(* PLC project Error Translations, Hydac Systems GmbH PdtCodeBuilder.dll 1.2.7.80 *)
(* stored: companyURL http://www.hydac.com/, contentDescription This content was automatically generated. Please do not edit., creationDateTime 2025-04-18T16:40:50.760 *)

TYPE _eDm1ErrorText : (txt_Err_Spn1000_Fmi31_FmiExt255 := 0, txt_Err_Spn1001_Fmi31_FmiExt255 := 1, txt_Err_Spn1002_Fmi31_FmiExt255 := 2, txt_Err_Spn1003_Fmi31_FmiExt255 := 3, txt_Err_Spn1004_Fmi31_FmiExt255 := 4, txt_Err_Spn1005_Fmi31_FmiExt255 := 5, txt_Err_Spn1006_Fmi31_FmiExt255 := 6, txt_Err_Spn1007_Fmi31_FmiExt255 := 7, txt_Err_Spn1008_Fmi31_FmiExt255 := 8, txt_Err_Spn1009_Fmi31_FmiExt255 := 9, txt_Err_Spn1010_Fmi31_FmiExt255 := 10, txt_Err_Spn1011_Fmi31_FmiExt255 := 11, txt_Err_Spn1012_Fmi31_FmiExt255 := 12, txt_Err_Spn1013_Fmi31_FmiExt255 := 13, txt_Err_Spn1014_Fmi31_FmiExt255 := 14, txt_Err_Spn1015_Fmi31_FmiExt255 := 15, txt_Err_Spn1016_Fmi31_FmiExt255 := 16, txt_Err_Spn1017_Fmi31_FmiExt255 := 17, txt_Err_Spn1018_Fmi31_FmiExt255 := 18, txt_Err_Spn1019_Fmi31_FmiExt255 := 19, txt_Err_Spn1020_Fmi31_FmiExt255 := 20, txt_Err_Spn1021_Fmi31_FmiExt255 := 21, txt_Err_Spn1022_Fmi31_FmiExt255 := 22, txt_Err_Spn1023_Fmi31_FmiExt255 := 23, txt_Err_Spn1024_Fmi31_FmiExt255 := 24, txt_Err_Spn1031_Fmi31_FmiExt255 := 25, txt_Err_Spn1032_Fmi31_FmiExt255 := 26, txt_Err_Spn1033_Fmi31_FmiExt255 := 27, txt_Err_Spn1034_Fmi31_FmiExt255 := 28, txt_Err_Spn1035_Fmi31_FmiExt255 := 29, txt_Err_Spn1036_Fmi31_FmiExt255 := 30, txt_Err_Spn1037_Fmi31_FmiExt255 := 31, txt_Err_Spn1038_Fmi31_FmiExt255 := 32, txt_Err_Spn1039_Fmi31_FmiExt255 := 33, txt_Err_Spn1040_Fmi31_FmiExt255 := 34, txt_Err_Spn1041_Fmi31_FmiExt255 := 35, txt_Err_Spn1042_Fmi31_FmiExt255 := 36, txt_Err_Spn1043_Fmi31_FmiExt255 := 37, txt_Err_Spn1044_Fmi31_FmiExt255 := 38, txt_Err_Spn1045_Fmi31_FmiExt255 := 39, txt_Err_Spn1046_Fmi31_FmiExt255 := 40, txt_Err_Spn1047_Fmi31_FmiExt255 := 41, txt_Err_Spn1048_Fmi31_FmiExt255 := 42, txt_Err_Spn1049_Fmi31_FmiExt255 := 43, txt_Err_Spn1051_Fmi31_FmiExt255 := 44, txt_Err_Spn1052_Fmi31_FmiExt255 := 45, txt_Err_Spn1053_Fmi31_FmiExt255 := 46, txt_Err_Spn1054_Fmi31_FmiExt255 := 47, txt_Err_Spn1055_Fmi31_FmiExt255 := 48, txt_Err_Spn1056_Fmi31_FmiExt255 := 49, txt_Err_Spn1057_Fmi31_FmiExt255 := 50, txt_Err_Spn1058_Fmi31_FmiExt255 := 51, txt_Err_Spn1059_Fmi31_FmiExt255 := 52, txt_Err_Spn1060_Fmi31_FmiExt255 := 53, txt_Err_Spn1063_Fmi31_FmiExt255 := 54, txt_Err_Spn1064_Fmi31_FmiExt255 := 55, txt_Err_Spn1065_Fmi31_FmiExt255 := 56, txt_Err_Spn1066_Fmi31_FmiExt255 := 57, txt_Err_Spn1067_Fmi31_FmiExt255 := 58, txt_Err_Spn1068_Fmi31_FmiExt255 := 59, txt_Err_Spn1069_Fmi31_FmiExt255 := 60, txt_Err_Spn1070_Fmi31_FmiExt255 := 61, txt_Err_Spn1071_Fmi31_FmiExt255 := 62, txt_Err_Spn1072_Fmi31_FmiExt255 := 63, txt_Err_Spn1073_Fmi31_FmiExt255 := 64, txt_Err_Spn1074_Fmi31_FmiExt255 := 65, txt_Err_Spn1075_Fmi31_FmiExt255 := 66, txt_Err_Spn1082_Fmi31_FmiExt255 := 67, txt_Err_Spn1083_Fmi31_FmiExt255 := 68, txt_Err_Spn1084_Fmi31_FmiExt255 := 69, txt_Err_Spn1102_Fmi31_FmiExt255 := 70, txt_Err_Spn1103_Fmi31_FmiExt255 := 71, txt_Err_Spn1104_Fmi31_FmiExt255 := 72, txt_Err_Spn1105_Fmi31_FmiExt255 := 73, txt_Err_Spn1106_Fmi31_FmiExt255 := 74, txt_Err_Spn1107_Fmi31_FmiExt255 := 75, txt_Err_Spn1108_Fmi31_FmiExt255 := 76, txt_Err_Spn1109_Fmi31_FmiExt255 := 77, txt_Err_Spn1110_Fmi31_FmiExt255 := 78, txt_Err_Spn1111_Fmi31_FmiExt255 := 79, txt_Err_Spn1112_Fmi31_FmiExt255 := 80, txt_Err_Spn1113_Fmi31_FmiExt255 := 81, txt_Err_Spn1114_Fmi31_FmiExt255 := 82, txt_Err_Spn1115_Fmi31_FmiExt255 := 83, txt_Err_Spn1116_Fmi31_FmiExt255 := 84, txt_Err_Spn1117_Fmi31_FmiExt255 := 85, txt_Err_Spn1118_Fmi31_FmiExt255 := 86, txt_Err_Spn1119_Fmi31_FmiExt255 := 87, txt_Err_Spn1153_Fmi31_FmiExt255 := 88, txt_Err_Spn1154_Fmi31_FmiExt255 := 89, txt_Err_Spn1155_Fmi31_FmiExt255 := 90, txt_Err_Spn1156_Fmi31_FmiExt255 := 91, txt_Err_Spn1157_Fmi31_FmiExt255 := 92, txt_Err_Spn1158_Fmi31_FmiExt255 := 93, txt_Err_Spn1159_Fmi31_FmiExt255 := 94, txt_Err_Spn1160_Fmi31_FmiExt255 := 95, txt_Err_Spn1161_Fmi31_FmiExt255 := 96, txt_Err_Spn1162_Fmi31_FmiExt255 := 97, txt_Err_Spn1163_Fmi31_FmiExt255 := 98, txt_Err_Spn1164_Fmi31_FmiExt255 := 99, txt_Err_Spn1165_Fmi31_FmiExt255 := 100, txt_Err_Spn1166_Fmi31_FmiExt255 := 101, txt_Err_Spn1167_Fmi31_FmiExt255 := 102, txt_Err_Spn1168_Fmi31_FmiExt255 := 103, txt_Err_Spn1173_Fmi31_FmiExt255 := 104, txt_Err_Spn1174_Fmi31_FmiExt255 := 105, txt_Err_Spn1175_Fmi31_FmiExt255 := 106, txt_Err_Spn1176_Fmi31_FmiExt255 := 107, txt_Err_Spn1177_Fmi31_FmiExt255 := 108, txt_Err_Spn1178_Fmi31_FmiExt255 := 109, txt_Err_Spn1179_Fmi31_FmiExt255 := 110, txt_Err_Spn1180_Fmi31_FmiExt255 := 111, txt_Err_Spn1181_Fmi31_FmiExt255 := 112, txt_Err_Spn1182_Fmi31_FmiExt255 := 113, txt_Err_Spn1183_Fmi31_FmiExt255 := 114, txt_Err_Spn1184_Fmi31_FmiExt255 := 115, txt_Err_Spn1185_Fmi31_FmiExt255 := 116, txt_Err_Spn1186_Fmi31_FmiExt255 := 117, txt_Err_Spn1187_Fmi31_FmiExt255 := 118, txt_Err_Spn1188_Fmi31_FmiExt255 := 119, txt_Err_Spn1189_Fmi31_FmiExt255 := 120, txt_Err_Spn1190_Fmi31_FmiExt255 := 121, txt_Err_Spn1203_Fmi31_FmiExt255 := 122, txt_Err_Spn1205_Fmi31_FmiExt255 := 123, txt_Err_Spn1209_Fmi31_FmiExt255 := 124, txt_Err_Spn1210_Fmi31_FmiExt255 := 125, txt_Err_Spn1211_Fmi31_FmiExt255 := 126, txt_Err_Spn1212_Fmi31_FmiExt255 := 127, txt_Err_Spn1213_Fmi31_FmiExt255 := 128, txt_Err_Spn1214_Fmi31_FmiExt255 := 129, txt_Err_Spn1215_Fmi31_FmiExt255 := 130, txt_Err_Spn1216_Fmi31_FmiExt255 := 131, txt_Err_Spn1217_Fmi31_FmiExt255 := 132, txt_Err_Spn1218_Fmi31_FmiExt255 := 133, txt_Err_Spn1219_Fmi31_FmiExt255 := 134, txt_Err_Spn1220_Fmi31_FmiExt255 := 135, txt_Err_Spn1221_Fmi31_FmiExt255 := 136, txt_Err_Spn1222_Fmi31_FmiExt255 := 137, txt_Err_Spn1223_Fmi31_FmiExt255 := 138, txt_Err_Spn1224_Fmi31_FmiExt255 := 139, txt_Err_Spn1225_Fmi31_FmiExt255 := 140, txt_Err_Spn1226_Fmi31_FmiExt255 := 141, txt_Err_Spn1229_Fmi31_FmiExt255 := 142, txt_Err_Spn1230_Fmi31_FmiExt255 := 143, txt_Err_Spn1231_Fmi31_FmiExt255 := 144, txt_Err_Spn1232_Fmi31_FmiExt255 := 145, txt_Err_Spn1233_Fmi31_FmiExt255 := 146, txt_Err_Spn1234_Fmi31_FmiExt255 := 147, txt_Err_Spn1235_Fmi31_FmiExt255 := 148, txt_Err_Spn1236_Fmi31_FmiExt255 := 149, txt_Err_Spn1237_Fmi31_FmiExt255 := 150, txt_Err_Spn1238_Fmi31_FmiExt255 := 151, txt_Err_Spn1239_Fmi31_FmiExt255 := 152, txt_Err_Spn1240_Fmi31_FmiExt255 := 153, txt_Err_Spn1241_Fmi31_FmiExt255 := 154, txt_Err_Spn1242_Fmi31_FmiExt255 := 155, txt_Err_Spn1243_Fmi31_FmiExt255 := 156, txt_Err_Spn1244_Fmi31_FmiExt255 := 157, txt_Err_Spn1245_Fmi31_FmiExt255 := 158, txt_Err_Spn1246_Fmi31_FmiExt255 := 159, txt_Err_Spn1247_Fmi31_FmiExt255 := 160, txt_Err_Spn1253_Fmi31_FmiExt255 := 161, txt_Err_Spn1254_Fmi31_FmiExt255 := 162, txt_Err_Spn1255_Fmi31_FmiExt255 := 163, txt_Err_Spn1256_Fmi31_FmiExt255 := 164, txt_Err_Spn1257_Fmi31_FmiExt255 := 165, txt_Err_Spn1265_Fmi31_FmiExt255 := 166, txt_Err_Spn1266_Fmi31_FmiExt255 := 167, txt_Err_Spn1267_Fmi31_FmiExt255 := 168, txt_Err_Spn1268_Fmi31_FmiExt255 := 169, txt_Err_Spn1269_Fmi31_FmiExt255 := 170, txt_Err_Spn1277_Fmi31_FmiExt255 := 171, txt_Err_Spn1278_Fmi31_FmiExt255 := 172, txt_Err_Spn1279_Fmi31_FmiExt255 := 173, txt_Err_Spn1280_Fmi31_FmiExt255 := 174, txt_Err_Spn1281_Fmi31_FmiExt255 := 175, txt_Err_Spn1287_Fmi31_FmiExt255 := 176, txt_Err_Spn1288_Fmi31_FmiExt255 := 177, txt_Err_Spn1289_Fmi31_FmiExt255 := 178, txt_Err_Spn1290_Fmi31_FmiExt255 := 179, txt_Err_Spn1291_Fmi31_FmiExt255 := 180, txt_Err_Spn1292_Fmi31_FmiExt255 := 181, txt_Err_Spn1293_Fmi31_FmiExt255 := 182, txt_Err_Spn1294_Fmi31_FmiExt255 := 183, txt_Err_Spn1295_Fmi31_FmiExt255 := 184, txt_Err_Spn1296_Fmi31_FmiExt255 := 185, txt_Err_Spn1297_Fmi31_FmiExt255 := 186, txt_Err_Spn1298_Fmi31_FmiExt255 := 187, txt_Err_Spn1299_Fmi31_FmiExt255 := 188, txt_Err_Spn1300_Fmi31_FmiExt255 := 189, txt_Err_Spn1301_Fmi31_FmiExt255 := 190, txt_Err_Spn1302_Fmi31_FmiExt255 := 191, txt_Err_Spn1303_Fmi31_FmiExt255 := 192, txt_Err_Spn1304_Fmi31_FmiExt255 := 193, txt_Err_Spn1305_Fmi31_FmiExt255 := 194, txt_Err_Spn1306_Fmi31_FmiExt255 := 195, txt_Err_Spn1307_Fmi31_FmiExt255 := 196, txt_Err_Spn1308_Fmi31_FmiExt255 := 197, txt_Err_Spn1309_Fmi31_FmiExt255 := 198, txt_Err_Spn1310_Fmi31_FmiExt255 := 199, txt_Err_Spn1311_Fmi31_FmiExt255 := 200, txt_Err_Spn1312_Fmi31_FmiExt255 := 201, txt_Err_Spn1313_Fmi31_FmiExt255 := 202, txt_Err_Spn1314_Fmi31_FmiExt255 := 203, txt_Err_Spn1315_Fmi31_FmiExt255 := 204, txt_Err_Spn1316_Fmi31_FmiExt255 := 205, txt_Err_Spn1317_Fmi31_FmiExt255 := 206, txt_Err_Spn1318_Fmi31_FmiExt255 := 207, txt_Err_Spn1319_Fmi31_FmiExt255 := 208, txt_Err_Spn1320_Fmi31_FmiExt255 := 209, txt_Err_Spn1321_Fmi31_FmiExt255 := 210, txt_Err_Spn1322_Fmi31_FmiExt255 := 211, txt_Err_Spn1339_Fmi31_FmiExt255 := 212, txt_Err_Spn1345_Fmi31_FmiExt255 := 213, txt_Err_Spn1346_Fmi31_FmiExt255 := 214, txt_Err_Spn1347_Fmi31_FmiExt255 := 215, txt_Err_Spn1348_Fmi31_FmiExt255 := 216, txt_Err_Spn1349_Fmi31_FmiExt255 := 217, txt_Err_Spn1350_Fmi31_FmiExt255 := 218, txt_Err_Spn1351_Fmi31_FmiExt255 := 219, txt_Err_Spn1352_Fmi31_FmiExt255 := 220, txt_Err_Spn1353_Fmi31_FmiExt255 := 221, txt_Err_Spn1356_Fmi31_FmiExt255 := 222, txt_Err_Spn1357_Fmi31_FmiExt255 := 223, txt_Err_Spn1358_Fmi31_FmiExt255 := 224, txt_Err_Spn1359_Fmi31_FmiExt255 := 225, txt_Err_Spn1360_Fmi31_FmiExt255 := 226, txt_Err_Spn1361_Fmi31_FmiExt255 := 227, txt_Err_Spn1362_Fmi31_FmiExt255 := 228, txt_Err_Spn1363_Fmi31_FmiExt255 := 229, txt_Err_Spn1364_Fmi31_FmiExt255 := 230, txt_Err_Spn1365_Fmi31_FmiExt255 := 231, txt_Err_Spn1366_Fmi31_FmiExt255 := 232, txt_Err_Spn1367_Fmi31_FmiExt255 := 233, txt_Err_Spn1368_Fmi31_FmiExt255 := 234, txt_Err_Spn1369_Fmi31_FmiExt255 := 235, txt_Err_Spn1370_Fmi31_FmiExt255 := 236, txt_Err_Spn1371_Fmi31_FmiExt255 := 237, txt_Err_Spn1372_Fmi31_FmiExt255 := 238, txt_Err_Spn1373_Fmi31_FmiExt255 := 239, txt_Err_Spn1439_Fmi31_FmiExt255 := 240, txt_Err_Spn1440_Fmi31_FmiExt255 := 241, txt_Err_Spn1441_Fmi31_FmiExt255 := 242, txt_Err_Spn1442_Fmi31_FmiExt255 := 243, txt_Err_Spn1443_Fmi31_FmiExt255 := 244, txt_Err_Spn1449_Fmi31_FmiExt255 := 245, txt_Err_Spn1450_Fmi31_FmiExt255 := 246, txt_Err_Spn1451_Fmi31_FmiExt255 := 247, txt_Err_Spn1452_Fmi31_FmiExt255 := 248, txt_Err_Spn1453_Fmi31_FmiExt255 := 249, txt_Err_Spn1459_Fmi31_FmiExt255 := 250, txt_Err_Spn1460_Fmi31_FmiExt255 := 251, txt_Err_Spn1461_Fmi31_FmiExt255 := 252, txt_Err_Spn1462_Fmi31_FmiExt255 := 253, txt_Err_Spn1463_Fmi31_FmiExt255 := 254, txt_Err_Spn1469_Fmi31_FmiExt255 := 255, txt_Err_Spn1470_Fmi31_FmiExt255 := 256, txt_Err_Spn1471_Fmi31_FmiExt255 := 257, txt_Err_Spn1472_Fmi31_FmiExt255 := 258, txt_Err_Spn1473_Fmi31_FmiExt255 := 259, txt_Err_Spn1479_Fmi31_FmiExt255 := 260, txt_Err_Spn1480_Fmi31_FmiExt255 := 261, txt_Err_Spn1481_Fmi31_FmiExt255 := 262, txt_Err_Spn1482_Fmi31_FmiExt255 := 263, txt_Err_Spn1483_Fmi31_FmiExt255 := 264, txt_Err_Spn1536_Fmi31_FmiExt255 := 265, txt_Err_Spn1542_Fmi31_FmiExt255 := 266, txt_Err_Spn1543_Fmi31_FmiExt255 := 267, txt_Err_Spn1554_Fmi31_FmiExt255 := 268, txt_Err_Spn1566_Fmi31_FmiExt255 := 269, txt_Err_Spn1567_Fmi31_FmiExt255 := 270, txt_Err_Spn1568_Fmi31_FmiExt255 := 271, txt_Err_Spn1569_Fmi31_FmiExt255 := 272, txt_Err_Spn1570_Fmi31_FmiExt255 := 273, txt_Err_Spn1571_Fmi31_FmiExt255 := 274, txt_Err_Spn1572_Fmi31_FmiExt255 := 275, txt_Err_Spn1573_Fmi31_FmiExt255 := 276, txt_Err_Spn1574_Fmi31_FmiExt255 := 277, txt_Err_Spn1575_Fmi31_FmiExt255 := 278, txt_Err_Spn1576_Fmi31_FmiExt255 := 279, txt_Err_Spn1577_Fmi31_FmiExt255 := 280, txt_Err_Spn1578_Fmi31_FmiExt255 := 281, txt_Err_Spn1579_Fmi31_FmiExt255 := 282, txt_Err_Spn1580_Fmi31_FmiExt255 := 283, txt_Err_Spn1581_Fmi31_FmiExt255 := 284, txt_Err_Spn1582_Fmi31_FmiExt255 := 285, txt_Err_Spn1583_Fmi31_FmiExt255 := 286, txt_Err_Spn1584_Fmi31_FmiExt255 := 287, txt_Err_Spn1585_Fmi31_FmiExt255 := 288, txt_Err_Spn1586_Fmi31_FmiExt255 := 289, txt_Err_Spn1587_Fmi31_FmiExt255 := 290, txt_Err_Spn1588_Fmi31_FmiExt255 := 291, txt_Err_Spn1589_Fmi31_FmiExt255 := 292, txt_Err_Spn1590_Fmi31_FmiExt255 := 293, txt_Err_Spn1591_Fmi31_FmiExt255 := 294, txt_Err_Spn1592_Fmi31_FmiExt255 := 295, txt_Err_Spn1593_Fmi31_FmiExt255 := 296, txt_Err_Spn1594_Fmi31_FmiExt255 := 297, txt_Err_Spn1595_Fmi31_FmiExt255 := 298, txt_Err_Spn1596_Fmi31_FmiExt255 := 299, txt_Err_Spn1597_Fmi31_FmiExt255 := 300, txt_Err_Spn1598_Fmi31_FmiExt255 := 301, txt_Err_Spn9000_Fmi3_FmiExt255 := 302, txt_Err_Spn9001_Fmi4_FmiExt255 := 303, txt_Err_Spn9002_Fmi24_FmiExt255 := 304, txt_Err_Spn9003_Fmi12_FmiExt255 := 305, txt_Err_Spn9004_Fmi3_FmiExt255 := 306, txt_Err_Spn9005_Fmi4_FmiExt255 := 307, txt_Err_Spn9006_Fmi24_FmiExt255 := 308, txt_Err_Spn9007_Fmi12_FmiExt255 := 309, txt_Err_Spn9008_Fmi3_FmiExt255 := 310, txt_Err_Spn9009_Fmi4_FmiExt255 := 311, txt_Err_Spn9010_Fmi24_FmiExt255 := 312, txt_Err_Spn9011_Fmi12_FmiExt255 := 313, txt_Err_Spn9012_Fmi31_FmiExt255 := 314, txt_Err_Spn9013_Fmi31_FmiExt255 := 315, txt_Err_Spn9014_Fmi31_FmiExt255 := 316, txt_Err_Spn9015_Fmi31_FmiExt255 := 317, txt_Err_Spn9016_Fmi31_FmiExt255 := 318, txt_Err_Spn9017_Fmi31_FmiExt255 := 319, txt_Err_Spn9018_Fmi31_FmiExt255 := 320, txt_Err_Spn9019_Fmi31_FmiExt255 := 321, txt_Err_Spn9020_Fmi31_FmiExt255 := 322, txt_Err_Spn9021_Fmi31_FmiExt255 := 323, txt_Err_Spn9022_Fmi31_FmiExt255 := 324, txt_Err_Spn9023_Fmi31_FmiExt255 := 325, txt_Err_Spn9024_Fmi31_FmiExt255 := 326, txt_Err_Spn9025_Fmi31_FmiExt255 := 327, txt_Err_Spn9026_Fmi31_FmiExt255 := 328, txt_Err_Spn9027_Fmi31_FmiExt255 := 329, txt_Err_Spn9028_Fmi31_FmiExt255 := 330, txt_Err_Spn9029_Fmi31_FmiExt255 := 331, txt_Err_Spn9030_Fmi31_FmiExt255 := 332, txt_Err_Spn9031_Fmi31_FmiExt255 := 333, txt_Err_Spn9032_Fmi31_FmiExt255 := 334, txt_Err_Spn9033_Fmi31_FmiExt255 := 335, txt_Err_Spn9034_Fmi31_FmiExt255 := 336, txt_Err_Spn9035_Fmi31_FmiExt255 := 337, txt_Err_Spn9036_Fmi31_FmiExt255 := 338, txt_Err_Spn9037_Fmi31_FmiExt255 := 339, txt_Err_Spn9038_Fmi31_FmiExt255 := 340, txt_Err_Spn9039_Fmi31_FmiExt255 := 341, txt_Err_Spn9040_Fmi31_FmiExt255 := 342, txt_Err_Spn9041_Fmi31_FmiExt255 := 343, txt_Err_Spn9042_Fmi31_FmiExt255 := 344, txt_Err_Spn9043_Fmi31_FmiExt255 := 345, txt_Err_Spn9044_Fmi31_FmiExt255 := 346, txt_Err_Spn9045_Fmi31_FmiExt255 := 347, txt_Err_Spn9046_Fmi31_FmiExt255 := 348, txt_Err_Spn9047_Fmi31_FmiExt255 := 349, txt_Err_Spn9048_Fmi3_FmiExt255 := 350, txt_Err_Spn9049_Fmi4_FmiExt255 := 351, txt_Err_Spn9050_Fmi24_FmiExt255 := 352, txt_Err_Spn9051_Fmi12_FmiExt255 := 353, txt_Err_Spn9052_Fmi31_FmiExt255 := 354, txt_Err_Spn9053_Fmi31_FmiExt255 := 355, txt_Err_Spn9054_Fmi31_FmiExt255 := 356, txt_Err_Spn9055_Fmi31_FmiExt255 := 357, txt_Err_Spn9056_Fmi31_FmiExt255 := 358, txt_Err_Spn9057_Fmi31_FmiExt255 := 359, txt_Err_Spn9058_Fmi31_FmiExt255 := 360, txt_Err_Spn9059_Fmi31_FmiExt255 := 361, txt_Err_Spn9060_Fmi31_FmiExt255 := 362, txt_Err_Spn9061_Fmi31_FmiExt255 := 363, txt_Err_Spn9062_Fmi31_FmiExt255 := 364, txt_Err_Spn9063_Fmi31_FmiExt255 := 365, txt_Err_Spn9064_Fmi3_FmiExt255 := 366, txt_Err_Spn9065_Fmi4_FmiExt255 := 367, txt_Err_Spn9066_Fmi24_FmiExt255 := 368, txt_Err_Spn9067_Fmi12_FmiExt255 := 369, txt_Err_Spn9068_Fmi31_FmiExt255 := 370, txt_Err_Spn9069_Fmi31_FmiExt255 := 371, txt_Err_Spn9070_Fmi31_FmiExt255 := 372, txt_Err_Spn9071_Fmi31_FmiExt255 := 373, txt_Err_Spn9072_Fmi31_FmiExt255 := 374, txt_Err_Spn9073_Fmi31_FmiExt255 := 375, txt_Err_Spn9074_Fmi31_FmiExt255 := 376, txt_Err_Spn9075_Fmi31_FmiExt255 := 377, txt_Err_Spn9076_Fmi31_FmiExt255 := 378, txt_Err_Spn9077_Fmi31_FmiExt255 := 379, txt_Err_Spn9078_Fmi31_FmiExt255 := 380, txt_Err_Spn9079_Fmi31_FmiExt255 := 381, txt_Err_Spn9080_Fmi31_FmiExt255 := 382, txt_Err_Spn9081_Fmi31_FmiExt255 := 383, txt_Err_Spn9082_Fmi31_FmiExt255 := 384, txt_Err_Spn9083_Fmi31_FmiExt255 := 385, txt_Err_Spn9084_Fmi31_FmiExt255 := 386, txt_Err_Spn9085_Fmi31_FmiExt255 := 387, txt_Err_Spn9086_Fmi31_FmiExt255 := 388, txt_Err_Spn9087_Fmi31_FmiExt255 := 389, txt_Err_Spn9088_Fmi31_FmiExt255 := 390, txt_Err_Spn9089_Fmi31_FmiExt255 := 391, txt_Err_Spn9090_Fmi31_FmiExt255 := 392, txt_Err_Spn9091_Fmi31_FmiExt255 := 393, txt_Err_Spn9092_Fmi31_FmiExt255 := 394, txt_Err_Spn9093_Fmi31_FmiExt255 := 395, txt_Err_Spn9094_Fmi31_FmiExt255 := 396, txt_Err_Spn9095_Fmi31_FmiExt255 := 397, txt_Err_Spn9096_Fmi31_FmiExt255 := 398, txt_Err_Spn9097_Fmi31_FmiExt255 := 399, txt_Err_Spn9098_Fmi31_FmiExt255 := 400, txt_Err_Spn9099_Fmi31_FmiExt255 := 401, txt_Err_Spn9100_Fmi31_FmiExt255 := 402, txt_Err_Spn9101_Fmi31_FmiExt255 := 403, txt_Err_Spn9102_Fmi31_FmiExt255 := 404, txt_Err_Spn9103_Fmi31_FmiExt255 := 405, txt_Err_Spn9104_Fmi31_FmiExt255 := 406, txt_Err_Spn9105_Fmi31_FmiExt255 := 407, txt_Err_Spn9106_Fmi31_FmiExt255 := 408, txt_Err_Spn9107_Fmi31_FmiExt255 := 409, txt_Err_Spn9108_Fmi31_FmiExt255 := 410, txt_Err_Spn9109_Fmi31_FmiExt255 := 411, txt_Err_Spn9110_Fmi31_FmiExt255 := 412, txt_Err_Spn9111_Fmi31_FmiExt255 := 413, txt_Err_Spn9112_Fmi31_FmiExt255 := 414, txt_Err_Spn9113_Fmi31_FmiExt255 := 415, txt_Err_Spn9114_Fmi31_FmiExt255 := 416, txt_Err_Spn9115_Fmi31_FmiExt255 := 417, txt_Err_Spn9116_Fmi31_FmiExt255 := 418, txt_Err_Spn9117_Fmi31_FmiExt255 := 419, txt_Err_Spn9118_Fmi31_FmiExt255 := 420, txt_Err_Spn9119_Fmi31_FmiExt255 := 421, txt_Err_Spn9120_Fmi31_FmiExt255 := 422, txt_Err_Spn9121_Fmi31_FmiExt255 := 423, txt_Err_Spn9122_Fmi31_FmiExt255 := 424, txt_Err_Spn9123_Fmi31_FmiExt255 := 425, txt_Err_Spn9124_Fmi31_FmiExt255 := 426, txt_Err_Spn9125_Fmi31_FmiExt255 := 427, txt_Err_Spn9126_Fmi31_FmiExt255 := 428, txt_Err_Spn9127_Fmi31_FmiExt255 := 429, txt_Err_Spn9128_Fmi31_FmiExt255 := 430, txt_Err_Spn9129_Fmi31_FmiExt255 := 431, txt_Err_Spn9130_Fmi31_FmiExt255 := 432, txt_Err_Spn9131_Fmi31_FmiExt255 := 433, txt_Err_Spn9132_Fmi31_FmiExt255 := 434, txt_Err_Spn9133_Fmi31_FmiExt255 := 435, txt_Err_Spn9134_Fmi31_FmiExt255 := 436, txt_Err_Spn9135_Fmi31_FmiExt255 := 437, txt_Err_Spn9136_Fmi31_FmiExt255 := 438, txt_Err_Spn9137_Fmi31_FmiExt255 := 439, txt_Err_Spn9138_Fmi31_FmiExt255 := 440, txt_Err_Spn9139_Fmi31_FmiExt255 := 441, txt_Err_Spn9140_Fmi31_FmiExt255 := 442, txt_Err_Spn9141_Fmi31_FmiExt255 := 443, txt_Err_Spn9142_Fmi31_FmiExt255 := 444, txt_Err_Spn9143_Fmi31_FmiExt255 := 445, txt_Err_Spn9144_Fmi31_FmiExt255 := 446, txt_Err_Spn9145_Fmi31_FmiExt255 := 447, txt_Err_Spn9146_Fmi31_FmiExt255 := 448, txt_Err_Spn9147_Fmi31_FmiExt255 := 449, txt_Err_Spn9148_Fmi31_FmiExt255 := 450, txt_Err_Spn9149_Fmi31_FmiExt255 := 451, txt_Err_Spn9150_Fmi31_FmiExt255 := 452, txt_Err_Spn9151_Fmi31_FmiExt255 := 453, txt_Err_Spn9152_Fmi31_FmiExt255 := 454, txt_Err_Spn9153_Fmi31_FmiExt255 := 455, txt_Err_Spn9154_Fmi31_FmiExt255 := 456, txt_Err_Spn9155_Fmi31_FmiExt255 := 457, txt_Err_Spn9156_Fmi31_FmiExt255 := 458, txt_Err_Spn9157_Fmi31_FmiExt255 := 459, txt_Err_Spn9158_Fmi31_FmiExt255 := 460, txt_Err_Spn9159_Fmi31_FmiExt255 := 461, txt_Err_Spn9160_Fmi31_FmiExt255 := 462, txt_Err_Spn9161_Fmi31_FmiExt255 := 463, txt_Err_Spn9162_Fmi31_FmiExt255 := 464, txt_Err_Spn9163_Fmi31_FmiExt255 := 465, txt_Err_Spn9164_Fmi31_FmiExt255 := 466, txt_Err_Spn9165_Fmi31_FmiExt255 := 467, txt_Err_Spn9166_Fmi31_FmiExt255 := 468, txt_Err_Spn9167_Fmi31_FmiExt255 := 469, txt_Err_Spn9168_Fmi31_FmiExt255 := 470, txt_Err_Spn9169_Fmi31_FmiExt255 := 471, txt_Err_Spn9170_Fmi31_FmiExt255 := 472, txt_Err_Spn9171_Fmi31_FmiExt255 := 473, txt_Err_Spn9172_Fmi31_FmiExt255 := 474, txt_Err_Spn9173_Fmi3_FmiExt255 := 475, txt_Err_Spn9174_Fmi4_FmiExt255 := 476, txt_Err_Spn9175_Fmi24_FmiExt255 := 477, txt_Err_Spn9176_Fmi12_FmiExt255 := 478, txt_Err_Spn9177_Fmi31_FmiExt255 := 479, txt_Err_Spn9178_Fmi31_FmiExt255 := 480, txt_Err_Spn9179_Fmi31_FmiExt255 := 481, txt_Err_Spn9180_Fmi31_FmiExt255 := 482, txt_Err_Spn9181_Fmi31_FmiExt255 := 483, txt_Err_Spn9182_Fmi31_FmiExt255 := 484, txt_Err_Spn9183_Fmi31_FmiExt255 := 485, txt_Err_Spn9184_Fmi31_FmiExt255 := 486, txt_Err_Spn9185_Fmi31_FmiExt255 := 487, txt_Err_Spn9186_Fmi31_FmiExt255 := 488, txt_Err_Spn9187_Fmi31_FmiExt255 := 489, txt_Err_Spn9188_Fmi31_FmiExt255 := 490, txt_Err_Spn9189_Fmi31_FmiExt255 := 491, txt_Err_Spn9190_Fmi31_FmiExt255 := 492, txt_Err_Spn9191_Fmi31_FmiExt255 := 493, txt_Err_Spn9192_Fmi31_FmiExt255 := 494, txt_Err_Spn9193_Fmi31_FmiExt255 := 495, txt_Err_Spn9194_Fmi31_FmiExt255 := 496, txt_Err_Spn9195_Fmi31_FmiExt255 := 497, txt_Err_Spn9196_Fmi31_FmiExt255 := 498, txt_Err_Spn9197_Fmi31_FmiExt255 := 499, txt_Err_Spn9198_Fmi31_FmiExt255 := 500, txt_Err_Spn9199_Fmi31_FmiExt255 := 501, txt_Err_Spn9200_Fmi31_FmiExt255 := 502, txt_Err_Spn9201_Fmi31_FmiExt255 := 503, txt_Err_Spn9202_Fmi31_FmiExt255 := 504, txt_Err_Spn9203_Fmi31_FmiExt255 := 505, txt_Err_Spn9204_Fmi31_FmiExt255 := 506, txt_Err_Spn9205_Fmi31_FmiExt255 := 507, txt_Err_Spn9206_Fmi31_FmiExt255 := 508, txt_Err_Spn9207_Fmi31_FmiExt255 := 509, txt_Err_Spn9208_Fmi31_FmiExt255 := 510, txt_Err_Spn9209_Fmi31_FmiExt255 := 511, txt_Err_Spn9210_Fmi31_FmiExt255 := 512, txt_Err_Spn9211_Fmi31_FmiExt255 := 513, txt_Err_Spn9212_Fmi31_FmiExt255 := 514, txt_Err_Spn9213_Fmi31_FmiExt255 := 515, txt_Err_Spn9214_Fmi31_FmiExt255 := 516, txt_Err_Spn9215_Fmi31_FmiExt255 := 517, txt_Err_Spn9216_Fmi31_FmiExt255 := 518, txt_Err_Spn9217_Fmi31_FmiExt255 := 519, txt_Err_Spn9218_Fmi31_FmiExt255 := 520, txt_Err_Spn9219_Fmi31_FmiExt255 := 521, txt_Err_Spn9220_Fmi31_FmiExt255 := 522, txt_Err_Spn9221_Fmi31_FmiExt255 := 523, txt_Err_Spn9222_Fmi31_FmiExt255 := 524, txt_Err_Spn9223_Fmi31_FmiExt255 := 525, txt_Err_Spn9224_Fmi31_FmiExt255 := 526, txt_Err_Spn9225_Fmi31_FmiExt255 := 527, txt_Err_Spn9226_Fmi31_FmiExt255 := 528, txt_Err_Spn9227_Fmi31_FmiExt255 := 529, txt_Err_Spn9228_Fmi31_FmiExt255 := 530, txt_Err_Spn9237_Fmi31_FmiExt255 := 531, txt_Err_Spn9238_Fmi31_FmiExt255 := 532, txt_Err_Spn9239_Fmi31_FmiExt255 := 533, txt_Err_Spn9240_Fmi31_FmiExt255 := 534, txt_Err_Spn9241_Fmi31_FmiExt255 := 535, txt_Err_Spn9242_Fmi31_FmiExt255 := 536, txt_Err_Spn9243_Fmi31_FmiExt255 := 537, txt_Err_Spn9244_Fmi31_FmiExt255 := 538, txt_Err_Spn9245_Fmi31_FmiExt255 := 539, txt_Err_Spn9246_Fmi3_FmiExt255 := 540, txt_Err_Spn9247_Fmi4_FmiExt255 := 541, txt_Err_Spn9248_Fmi24_FmiExt255 := 542, txt_Err_Spn9249_Fmi12_FmiExt255 := 543, txt_Err_Spn9250_Fmi3_FmiExt255 := 544, txt_Err_Spn9251_Fmi4_FmiExt255 := 545, txt_Err_Spn9252_Fmi24_FmiExt255 := 546, txt_Err_Spn9253_Fmi12_FmiExt255 := 547, txt_Err_Spn9254_Fmi31_FmiExt255 := 548, txt_Err_Spn9255_Fmi31_FmiExt255 := 549, txt_Err_Spn9256_Fmi31_FmiExt255 := 550, txt_Err_Spn9257_Fmi31_FmiExt255 := 551, txt_Err_Spn9258_Fmi31_FmiExt255 := 552, txt_Err_Spn9259_Fmi31_FmiExt255 := 553, txt_Err_Spn9260_Fmi31_FmiExt255 := 554, txt_Err_Spn9261_Fmi31_FmiExt255 := 555, txt_Err_Spn9262_Fmi31_FmiExt255 := 556, txt_Err_Spn9263_Fmi31_FmiExt255 := 557, txt_Err_Spn9264_Fmi31_FmiExt255 := 558, txt_Err_Spn9265_Fmi31_FmiExt255 := 559, txt_Err_Spn9266_Fmi31_FmiExt255 := 560, txt_Err_Spn9267_Fmi31_FmiExt255 := 561, txt_Err_Spn9268_Fmi31_FmiExt255 := 562, txt_Err_Spn9269_Fmi31_FmiExt255 := 563, txt_Err_Spn9270_Fmi31_FmiExt255 := 564, txt_Err_Spn9271_Fmi31_FmiExt255 := 565, txt_Err_Spn9272_Fmi31_FmiExt255 := 566, txt_Err_Spn9273_Fmi31_FmiExt255 := 567, txt_Err_Spn9274_Fmi31_FmiExt255 := 568, txt_Err_Spn9275_Fmi31_FmiExt255 := 569, txt_Err_Spn9276_Fmi31_FmiExt255 := 570, txt_Err_Spn9277_Fmi31_FmiExt255 := 571, txt_Err_Spn9278_Fmi31_FmiExt255 := 572, txt_Err_Spn9279_Fmi31_FmiExt255 := 573, txt_Err_Spn9280_Fmi31_FmiExt255 := 574, txt_Err_Spn9281_Fmi31_FmiExt255 := 575, txt_Err_Spn9282_Fmi31_FmiExt255 := 576, txt_Err_Spn9283_Fmi31_FmiExt255 := 577, txt_Err_Spn9284_Fmi31_FmiExt255 := 578, txt_Err_Spn9285_Fmi31_FmiExt255 := 579, txt_Err_Spn9286_Fmi31_FmiExt255 := 580, txt_Err_Spn9287_Fmi31_FmiExt255 := 581, txt_Err_Spn9288_Fmi31_FmiExt255 := 582, txt_Err_Spn9289_Fmi31_FmiExt255 := 583, txt_Err_Spn9290_Fmi31_FmiExt255 := 584, txt_Err_Spn9291_Fmi31_FmiExt255 := 585, txt_Err_Spn9292_Fmi31_FmiExt255 := 586, txt_Err_Spn9293_Fmi31_FmiExt255 := 587, txt_Err_Spn9294_Fmi31_FmiExt255 := 588, txt_Err_Spn9295_Fmi31_FmiExt255 := 589, txt_Err_Spn9296_Fmi31_FmiExt255 := 590, txt_Err_Spn9297_Fmi31_FmiExt255 := 591, txt_Err_Spn9298_Fmi31_FmiExt255 := 592, txt_Err_Spn9299_Fmi31_FmiExt255 := 593, txt_Err_Spn9300_Fmi31_FmiExt255 := 594, txt_Err_Spn9301_Fmi31_FmiExt255 := 595, txt_Err_Spn9302_Fmi31_FmiExt255 := 596, txt_Err_Spn9303_Fmi31_FmiExt255 := 597, txt_Err_Spn9304_Fmi31_FmiExt255 := 598, txt_Err_Spn9305_Fmi31_FmiExt255 := 599, txt_Err_Spn9306_Fmi31_FmiExt255 := 600, txt_Err_Spn9307_Fmi31_FmiExt255 := 601, txt_Err_Spn9308_Fmi31_FmiExt255 := 602, txt_Err_Spn9309_Fmi31_FmiExt255 := 603, txt_Err_Spn9310_Fmi31_FmiExt255 := 604, txt_Err_Spn9311_Fmi31_FmiExt255 := 605, txt_Err_Spn9312_Fmi31_FmiExt255 := 606, txt_Err_Spn9313_Fmi31_FmiExt255 := 607, txt_Err_Spn9314_Fmi31_FmiExt255 := 608, txt_Err_Spn9315_Fmi31_FmiExt255 := 609, txt_Err_Spn9316_Fmi31_FmiExt255 := 610, txt_Err_Spn9317_Fmi31_FmiExt255 := 611, txt_Err_Spn9318_Fmi31_FmiExt255 := 612, txt_Err_Spn9319_Fmi31_FmiExt255 := 613, txt_Err_Spn9320_Fmi31_FmiExt255 := 614, txt_Err_Spn9321_Fmi31_FmiExt255 := 615, txt_Err_Spn9322_Fmi31_FmiExt255 := 616, txt_Err_Spn9323_Fmi31_FmiExt255 := 617, txt_Err_Spn9324_Fmi31_FmiExt255 := 618, txt_Err_Spn9325_Fmi31_FmiExt255 := 619, txt_Err_Spn9326_Fmi31_FmiExt255 := 620, txt_Err_Spn9327_Fmi31_FmiExt255 := 621, txt_Err_Spn9328_Fmi31_FmiExt255 := 622, txt_Err_Spn9329_Fmi31_FmiExt255 := 623, txt_Err_Spn9330_Fmi31_FmiExt255 := 624, txt_Err_Spn9331_Fmi31_FmiExt255 := 625, txt_Err_Spn9332_Fmi31_FmiExt255 := 626, txt_Err_Spn9333_Fmi31_FmiExt255 := 627, txt_Err_Spn9334_Fmi31_FmiExt255 := 628, txt_Err_Spn9335_Fmi31_FmiExt255 := 629, txt_Err_Spn9336_Fmi31_FmiExt255 := 630, txt_Err_Spn9337_Fmi31_FmiExt255 := 631, txt_Err_Spn9338_Fmi31_FmiExt255 := 632, txt_Err_Spn9339_Fmi31_FmiExt255 := 633, txt_Err_Spn9340_Fmi31_FmiExt255 := 634, txt_Err_Spn9341_Fmi31_FmiExt255 := 635, txt_Err_Spn9342_Fmi31_FmiExt255 := 636, txt_Err_Spn9343_Fmi31_FmiExt255 := 637, txt_Err_Spn9344_Fmi31_FmiExt255 := 638, txt_Err_Spn9345_Fmi31_FmiExt255 := 639, txt_Err_Spn9346_Fmi31_FmiExt255 := 640, txt_Err_Spn9347_Fmi31_FmiExt255 := 641, txt_Err_Spn9348_Fmi31_FmiExt255 := 642, txt_Err_Spn9349_Fmi31_FmiExt255 := 643, txt_Err_Spn9350_Fmi31_FmiExt255 := 644, txt_Err_Spn9351_Fmi31_FmiExt255 := 645, txt_Err_Spn9374_Fmi31_FmiExt255 := 646, txt_Err_Spn9375_Fmi31_FmiExt255 := 647, txt_Err_Spn9376_Fmi31_FmiExt255 := 648, txt_Err_Spn9377_Fmi31_FmiExt255 := 649, txt_Err_Spn9378_Fmi31_FmiExt255 := 650, txt_Err_Spn9389_Fmi31_FmiExt255 := 651, txt_Err_Spn9390_Fmi31_FmiExt255 := 652, txt_Err_Spn9391_Fmi31_FmiExt255 := 653, txt_Err_Spn9392_Fmi31_FmiExt255 := 654, txt_Err_Spn9393_Fmi31_FmiExt255 := 655, txt_Err_Spn9394_Fmi31_FmiExt255 := 656, txt_Err_Spn9395_Fmi31_FmiExt255 := 657, txt_Err_Spn9396_Fmi31_FmiExt255 := 658, txt_Err_Spn9397_Fmi31_FmiExt255 := 659, txt_Err_Spn9398_Fmi31_FmiExt255 := 660, txt_Err_Spn9399_Fmi31_FmiExt255 := 661, txt_Err_Spn9400_Fmi31_FmiExt255 := 662, txt_Err_Spn9413_Fmi31_FmiExt255 := 663, txt_Err_Spn9414_Fmi31_FmiExt255 := 664, txt_Err_Spn9415_Fmi31_FmiExt255 := 665, txt_Err_Spn9416_Fmi31_FmiExt255 := 666, txt_Err_Spn9417_Fmi31_FmiExt255 := 667, txt_Err_Spn9418_Fmi31_FmiExt255 := 668, txt_Err_Spn9419_Fmi31_FmiExt255 := 669, txt_Err_Spn9437_Fmi31_FmiExt255 := 670, txt_Err_Spn9438_Fmi31_FmiExt255 := 671, txt_Err_Spn9439_Fmi31_FmiExt255 := 672, txt_Err_Spn9440_Fmi31_FmiExt255 := 673, txt_Err_Spn9441_Fmi31_FmiExt255 := 674, txt_Err_Spn9442_Fmi31_FmiExt255 := 675, txt_Err_Spn9443_Fmi31_FmiExt255 := 676, txt_Err_Spn9444_Fmi31_FmiExt255 := 677, txt_Err_Spn9445_Fmi31_FmiExt255 := 678, txt_Err_Spn9446_Fmi31_FmiExt255 := 679, txt_Err_Spn9447_Fmi31_FmiExt255 := 680, txt_Err_Spn9448_Fmi31_FmiExt255 := 681, txt_Err_Spn9449_Fmi31_FmiExt255 := 682, txt_Err_Spn9450_Fmi31_FmiExt255 := 683, txt_Err_Spn9451_Fmi31_FmiExt255 := 684, txt_Err_Spn9452_Fmi31_FmiExt255 := 685, txt_Err_Spn9479_Fmi31_FmiExt255 := 686, txt_Err_Spn9480_Fmi31_FmiExt255 := 687, txt_Err_Spn9481_Fmi31_FmiExt255 := 688, txt_Err_Spn9482_Fmi31_FmiExt255 := 689, txt_Err_Spn9483_Fmi31_FmiExt255 := 690, txt_Err_Spn9484_Fmi31_FmiExt255 := 691, txt_Err_Spn9485_Fmi31_FmiExt255 := 692, txt_Err_Spn9486_Fmi31_FmiExt255 := 693, txt_Err_Spn9487_Fmi31_FmiExt255 := 694, txt_Err_Spn9488_Fmi31_FmiExt255 := 695, txt_Err_Spn9489_Fmi31_FmiExt255 := 696, txt_Err_Spn9490_Fmi31_FmiExt255 := 697, txt_Err_Spn9491_Fmi31_FmiExt255 := 698, txt_Err_Spn9492_Fmi31_FmiExt255 := 699, txt_Err_Spn9493_Fmi31_FmiExt255 := 700, txt_Err_Spn9494_Fmi31_FmiExt255 := 701, txt_Err_Spn9495_Fmi31_FmiExt255 := 702, txt_Err_Spn9496_Fmi31_FmiExt255 := 703, txt_Err_Spn9497_Fmi31_FmiExt255 := 704, txt_Err_Spn9503_Fmi31_FmiExt255 := 705, txt_Err_Spn9504_Fmi31_FmiExt255 := 706, txt_Err_Spn9505_Fmi31_FmiExt255 := 707, txt_Err_Spn9506_Fmi31_FmiExt255 := 708, txt_Err_Spn9507_Fmi31_FmiExt255 := 709, txt_Err_Spn9508_Fmi31_FmiExt255 := 710, txt_Err_Spn9509_Fmi31_FmiExt255 := 711, txt_Err_Spn9510_Fmi31_FmiExt255 := 712, txt_Err_Spn9511_Fmi31_FmiExt255 := 713, txt_Err_Spn9512_Fmi31_FmiExt255 := 714, txt_Err_Spn9513_Fmi31_FmiExt255 := 715, txt_Err_Spn9514_Fmi31_FmiExt255 := 716, txt_Err_Spn9515_Fmi31_FmiExt255 := 717, txt_Err_Spn9516_Fmi31_FmiExt255 := 718, txt_Err_Spn9517_Fmi31_FmiExt255 := 719, txt_Err_Spn9523_Fmi31_FmiExt255 := 720, txt_Err_Spn9524_Fmi31_FmiExt255 := 721, txt_Err_Spn9525_Fmi31_FmiExt255 := 722, txt_Err_Spn9526_Fmi31_FmiExt255 := 723, txt_Err_Spn9527_Fmi31_FmiExt255 := 724, txt_Err_Spn9528_Fmi31_FmiExt255 := 725, txt_Err_Spn9529_Fmi31_FmiExt255 := 726, txt_Err_Spn9530_Fmi31_FmiExt255 := 727, txt_Err_Spn9531_Fmi31_FmiExt255 := 728, txt_Err_Spn9532_Fmi31_FmiExt255 := 729, txt_Err_Spn9533_Fmi31_FmiExt255 := 730, txt_Err_Spn9534_Fmi31_FmiExt255 := 731, txt_Err_Spn9535_Fmi31_FmiExt255 := 732, txt_Err_Spn9536_Fmi31_FmiExt255 := 733, txt_Err_Spn9537_Fmi31_FmiExt255 := 734, txt_Err_Spn9538_Fmi31_FmiExt255 := 735, txt_Err_Spn9539_Fmi31_FmiExt255 := 736, txt_Err_Spn9540_Fmi31_FmiExt255 := 737, txt_Err_Spn9541_Fmi31_FmiExt255 := 738, txt_Err_Spn9542_Fmi31_FmiExt255 := 739, txt_Err_Spn9543_Fmi31_FmiExt255 := 740, txt_Err_Spn9544_Fmi31_FmiExt255 := 741, txt_Err_Spn9545_Fmi31_FmiExt255 := 742, txt_Err_Spn9546_Fmi31_FmiExt255 := 743, txt_Err_Spn9547_Fmi31_FmiExt255 := 744, txt_Err_Spn9552_Fmi31_FmiExt255 := 745, txt_Err_Spn9553_Fmi31_FmiExt255 := 746, txt_Err_Spn9554_Fmi31_FmiExt255 := 747, txt_Err_Spn9555_Fmi31_FmiExt255 := 748, txt_Err_Spn9556_Fmi31_FmiExt255 := 749, txt_Err_Spn9557_Fmi31_FmiExt255 := 750, txt_Err_Spn9558_Fmi31_FmiExt255 := 751, txt_Err_Spn9559_Fmi31_FmiExt255 := 752, txt_Err_Spn9560_Fmi31_FmiExt255 := 753, txt_Err_Spn9561_Fmi31_FmiExt255 := 754, txt_Err_Spn9562_Fmi31_FmiExt255 := 755, txt_Err_Spn9563_Fmi31_FmiExt255 := 756, txt_Err_Spn9564_Fmi31_FmiExt255 := 757, txt_Err_Spn9565_Fmi31_FmiExt255 := 758, txt_Err_Spn9586_Fmi31_FmiExt255 := 759, txt_Err_Spn9587_Fmi31_FmiExt255 := 760, txt_Err_Spn9588_Fmi31_FmiExt255 := 761, txt_Err_Spn9589_Fmi31_FmiExt255 := 762, txt_Err_Spn9590_Fmi31_FmiExt255 := 763, txt_Err_Spn9591_Fmi31_FmiExt255 := 764, txt_Err_Spn9592_Fmi31_FmiExt255 := 765, txt_Err_Spn9593_Fmi31_FmiExt255 := 766, txt_Err_Spn9599_Fmi31_FmiExt255 := 767, txt_Err_Spn9600_Fmi31_FmiExt255 := 768, txt_Err_Spn9601_Fmi31_FmiExt255 := 769, txt_Err_Spn9602_Fmi31_FmiExt255 := 770, txt_Err_Spn9603_Fmi31_FmiExt255 := 771, txt_Err_Spn9604_Fmi31_FmiExt255 := 772, txt_Err_Spn9605_Fmi31_FmiExt255 := 773, txt_Err_Spn9606_Fmi31_FmiExt255 := 774, txt_Err_Spn9607_Fmi31_FmiExt255 := 775, txt_Err_Spn9608_Fmi31_FmiExt255 := 776, txt_Err_Spn9609_Fmi31_FmiExt255 := 777, txt_Err_Spn9610_Fmi31_FmiExt255 := 778, txt_Err_Spn9611_Fmi31_FmiExt255 := 779, txt_Err_Spn9612_Fmi31_FmiExt255 := 780, txt_Err_Spn9613_Fmi31_FmiExt255 := 781, txt_Err_Spn9614_Fmi31_FmiExt255 := 782, txt_Err_Spn9615_Fmi31_FmiExt255 := 783, txt_Err_Spn9616_Fmi31_FmiExt255 := 784, txt_Err_Spn9617_Fmi31_FmiExt255 := 785, txt_Err_Spn9618_Fmi31_FmiExt255 := 786, txt_Err_Spn9619_Fmi31_FmiExt255 := 787, txt_Err_Spn9620_Fmi31_FmiExt255 := 788, txt_Err_Spn9621_Fmi31_FmiExt255 := 789, txt_Err_Spn9622_Fmi31_FmiExt255 := 790, txt_Err_Spn9623_Fmi31_FmiExt255 := 791, txt_Err_Spn9624_Fmi31_FmiExt255 := 792, txt_Err_Spn9625_Fmi31_FmiExt255 := 793, txt_Err_Spn9626_Fmi31_FmiExt255 := 794, txt_Err_Spn9627_Fmi31_FmiExt255 := 795, txt_Err_Spn9628_Fmi31_FmiExt255 := 796, txt_Err_Spn9633_Fmi31_FmiExt255 := 797, txt_Err_Spn9634_Fmi31_FmiExt255 := 798, txt_Err_Spn9635_Fmi31_FmiExt255 := 799, txt_Err_Spn9636_Fmi31_FmiExt255 := 800, txt_Err_Spn9637_Fmi31_FmiExt255 := 801, txt_Err_Spn9638_Fmi31_FmiExt255 := 802, txt_Err_Spn9639_Fmi31_FmiExt255 := 803, txt_Err_Spn9640_Fmi31_FmiExt255 := 804, txt_Err_Spn9641_Fmi31_FmiExt255 := 805, txt_Err_Spn9642_Fmi31_FmiExt255 := 806, txt_Err_Spn9643_Fmi31_FmiExt255 := 807, txt_Err_Spn9644_Fmi31_FmiExt255 := 808, txt_Err_Spn9645_Fmi31_FmiExt255 := 809, txt_Err_Spn9646_Fmi31_FmiExt255 := 810, txt_Err_Spn9647_Fmi31_FmiExt255 := 811, txt_Err_Spn9648_Fmi31_FmiExt255 := 812, txt_Err_Spn9649_Fmi31_FmiExt255 := 813, txt_Err_Spn9650_Fmi31_FmiExt255 := 814, txt_Err_Spn9651_Fmi31_FmiExt255 := 815, txt_Err_Spn9652_Fmi31_FmiExt255 := 816, txt_Err_Spn9653_Fmi31_FmiExt255 := 817, txt_Err_Spn9654_Fmi31_FmiExt255 := 818, txt_Err_Spn9655_Fmi31_FmiExt255 := 819, txt_Err_Spn9656_Fmi31_FmiExt255 := 820, txt_Err_Spn9657_Fmi31_FmiExt255 := 821, txt_Err_Spn9658_Fmi31_FmiExt255 := 822, txt_Err_Spn9659_Fmi31_FmiExt255 := 823, txt_Err_Spn9660_Fmi31_FmiExt255 := 824, txt_Err_Spn9661_Fmi31_FmiExt255 := 825, txt_Err_Spn9662_Fmi31_FmiExt255 := 826, txt_Err_Spn9663_Fmi31_FmiExt255 := 827, txt_Err_Spn9664_Fmi31_FmiExt255 := 828, txt_Err_Spn9665_Fmi31_FmiExt255 := 829, txt_Err_Spn9666_Fmi31_FmiExt255 := 830, txt_Err_Spn9667_Fmi31_FmiExt255 := 831, txt_Err_Spn9668_Fmi31_FmiExt255 := 832, txt_Err_Spn9669_Fmi31_FmiExt255 := 833, txt_Err_Spn9670_Fmi31_FmiExt255 := 834, txt_Err_Spn9671_Fmi31_FmiExt255 := 835, txt_Err_Spn9672_Fmi31_FmiExt255 := 836, txt_Err_Spn9673_Fmi31_FmiExt255 := 837, txt_Err_Spn9674_Fmi31_FmiExt255 := 838, txt_Err_Spn9675_Fmi31_FmiExt255 := 839, txt_Err_Spn9676_Fmi31_FmiExt255 := 840, txt_Err_Spn9677_Fmi31_FmiExt255 := 841, txt_Err_Spn9678_Fmi31_FmiExt255 := 842, txt_Err_Spn9679_Fmi31_FmiExt255 := 843, txt_Err_Spn9680_Fmi31_FmiExt255 := 844, txt_Err_Spn9681_Fmi31_FmiExt255 := 845, txt_Err_Spn9682_Fmi31_FmiExt255 := 846, txt_Err_Spn9683_Fmi31_FmiExt255 := 847, txt_Err_Spn9684_Fmi31_FmiExt255 := 848, txt_Err_Spn9685_Fmi31_FmiExt255 := 849, txt_Err_Spn9686_Fmi31_FmiExt255 := 850, txt_Err_Spn9687_Fmi31_FmiExt255 := 851, txt_Err_Spn9688_Fmi31_FmiExt255 := 852, txt_Err_Spn9689_Fmi31_FmiExt255 := 853, txt_Err_Spn9690_Fmi31_FmiExt255 := 854, txt_Err_Spn9691_Fmi31_FmiExt255 := 855, txt_Err_Spn9692_Fmi31_FmiExt255 := 856, txt_Err_Spn9693_Fmi31_FmiExt255 := 857, txt_Err_Spn9694_Fmi31_FmiExt255 := 858, txt_Err_Spn9695_Fmi31_FmiExt255 := 859, txt_Err_Spn9696_Fmi31_FmiExt255 := 860, txt_Err_Spn9697_Fmi31_FmiExt255 := 861, txt_Err_Spn9698_Fmi31_FmiExt255 := 862, txt_Err_Spn9699_Fmi31_FmiExt255 := 863, txt_Err_Spn9700_Fmi31_FmiExt255 := 864, txt_Err_Spn9701_Fmi31_FmiExt255 := 865, txt_Err_Spn9702_Fmi31_FmiExt255 := 866, txt_Err_Spn9703_Fmi31_FmiExt255 := 867, txt_Err_Spn9704_Fmi31_FmiExt255 := 868, txt_Err_Spn9705_Fmi31_FmiExt255 := 869, txt_Err_Spn9706_Fmi31_FmiExt255 := 870, txt_Err_Spn9707_Fmi31_FmiExt255 := 871, txt_Err_Spn9708_Fmi31_FmiExt255 := 872, txt_Err_Spn9709_Fmi31_FmiExt255 := 873, txt_Err_Spn9710_Fmi31_FmiExt255 := 874, txt_Err_Spn9711_Fmi31_FmiExt255 := 875, txt_Err_Spn9712_Fmi31_FmiExt255 := 876, txt_Err_Spn9713_Fmi31_FmiExt255 := 877, txt_Err_Spn9714_Fmi31_FmiExt255 := 878, txt_Err_Spn9715_Fmi31_FmiExt255 := 879, txt_Err_Spn9716_Fmi31_FmiExt255 := 880, txt_Err_Spn9717_Fmi31_FmiExt255 := 881, txt_Err_Spn9718_Fmi31_FmiExt255 := 882, txt_Err_Spn9719_Fmi31_FmiExt255 := 883, txt_Err_Spn9720_Fmi31_FmiExt255 := 884, txt_Err_Spn9721_Fmi31_FmiExt255 := 885, txt_Err_Spn9722_Fmi31_FmiExt255 := 886, txt_Err_Spn9723_Fmi31_FmiExt255 := 887, txt_Err_Spn9724_Fmi31_FmiExt255 := 888, txt_Err_Spn9725_Fmi31_FmiExt255 := 889, txt_Err_Spn9726_Fmi31_FmiExt255 := 890, txt_Err_Spn9727_Fmi31_FmiExt255 := 891, txt_Err_Spn9732_Fmi31_FmiExt255 := 892, txt_Err_Spn9733_Fmi31_FmiExt255 := 893, txt_Err_Spn9734_Fmi31_FmiExt255 := 894, txt_Err_Spn9735_Fmi31_FmiExt255 := 895, txt_Err_Spn9756_Fmi3_FmiExt255 := 896, txt_Err_Spn9757_Fmi4_FmiExt255 := 897, txt_Err_Spn9758_Fmi3_FmiExt255 := 898, txt_Err_Spn9759_Fmi4_FmiExt255 := 899, txt_Err_Spn9760_Fmi26_FmiExt255 := 900, txt_Err_Spn9761_Fmi14_FmiExt255 := 901, txt_Err_Spn9762_Fmi24_FmiExt255 := 902, txt_Err_Spn9763_Fmi12_FmiExt255 := 903, txt_Err_Spn9764_Fmi3_FmiExt255 := 904, txt_Err_Spn9765_Fmi4_FmiExt255 := 905, txt_Err_Spn9766_Fmi3_FmiExt255 := 906, txt_Err_Spn9767_Fmi4_FmiExt255 := 907, txt_Err_Spn9768_Fmi26_FmiExt255 := 908, txt_Err_Spn9769_Fmi14_FmiExt255 := 909, txt_Err_Spn9770_Fmi24_FmiExt255 := 910, txt_Err_Spn9771_Fmi12_FmiExt255 := 911, txt_Err_Spn9772_Fmi31_FmiExt255 := 912, txt_Err_Spn9773_Fmi31_FmiExt255 := 913, txt_Err_Spn9774_Fmi31_FmiExt255 := 914, txt_Err_Spn9775_Fmi31_FmiExt255 := 915, txt_Err_Spn9776_Fmi31_FmiExt255 := 916, txt_Err_Spn9777_Fmi31_FmiExt255 := 917, txt_Err_Spn9778_Fmi31_FmiExt255 := 918, txt_Err_Spn9779_Fmi31_FmiExt255 := 919, txt_Err_Spn9780_Fmi31_FmiExt255 := 920, txt_Err_Spn15926_Fmi31_FmiExt255 := 921, txt_Err_Spn15927_Fmi31_FmiExt255 := 922, txt_Err_Spn15928_Fmi31_FmiExt255 := 923, txt_Err_Spn15929_Fmi31_FmiExt255 := 924, txt_Err_Spn15930_Fmi31_FmiExt255 := 925, txt_Err_Spn15931_Fmi31_FmiExt255 := 926, txt_Err_Spn15932_Fmi31_FmiExt255 := 927, txt_Err_Spn15933_Fmi31_FmiExt255 := 928, txt_Err_Spn15934_Fmi31_FmiExt255 := 929, txt_Err_Spn15935_Fmi31_FmiExt255 := 930, txt_Err_Spn15936_Fmi31_FmiExt255 := 931, txt_Err_Spn15941_Fmi31_FmiExt255 := 932, txt_Err_Spn15942_Fmi31_FmiExt255 := 933, txt_Err_Spn15943_Fmi31_FmiExt255 := 934, txt_Err_Spn15944_Fmi31_FmiExt255 := 935, txt_Err_Spn15945_Fmi31_FmiExt255 := 936, txt_Err_Spn15946_Fmi31_FmiExt255 := 937, txt_Err_Spn15947_Fmi31_FmiExt255 := 938, txt_Err_Spn15948_Fmi31_FmiExt255 := 939, txt_Err_Spn15949_Fmi31_FmiExt255 := 940, txt_Err_Spn15950_Fmi31_FmiExt255 := 941, txt_Err_Spn15951_Fmi31_FmiExt255 := 942, txt_Err_Spn15952_Fmi31_FmiExt255 := 943, txt_Err_Spn15953_Fmi31_FmiExt255 := 944, txt_Err_Spn15954_Fmi31_FmiExt255 := 945, txt_Err_Spn15955_Fmi31_FmiExt255 := 946, txt_Err_Spn15956_Fmi31_FmiExt255 := 947, txt_Err_Spn15973_Fmi31_FmiExt255 := 948, txt_Err_Spn15975_Fmi31_FmiExt255 := 949, txt_Err_Spn15976_Fmi31_FmiExt255 := 950, txt_Err_Spn15977_Fmi31_FmiExt255 := 951, txt_Err_Spn15978_Fmi31_FmiExt255 := 952, txt_Err_Spn15998_Fmi31_FmiExt255 := 953, txt_Err_Spn16004_Fmi31_FmiExt255 := 954, txt_Err_Spn16009_Fmi31_FmiExt255 := 955, txt_Err_Spn16014_Fmi31_FmiExt255 := 956, txt_Err_Spn16019_Fmi31_FmiExt255 := 957, txt_Err_Spn16024_Fmi31_FmiExt255 := 958, txt_Err_Spn16025_Fmi31_FmiExt255 := 959, txt_Err_Spn16026_Fmi31_FmiExt255 := 960, txt_Err_Spn16028_Fmi31_FmiExt255 := 961, txt_Err_Spn16029_Fmi31_FmiExt255 := 962, txt_Err_Spn16030_Fmi31_FmiExt255 := 963, txt_Err_Spn16031_Fmi31_FmiExt255 := 964, txt_Err_Spn16033_Fmi31_FmiExt255 := 965, txt_Err_Spn16034_Fmi31_FmiExt255 := 966, txt_Err_Spn16035_Fmi31_FmiExt255 := 967, txt_Err_Spn16036_Fmi31_FmiExt255 := 968, txt_Err_Spn16038_Fmi31_FmiExt255 := 969, txt_Err_Spn16042_Fmi31_FmiExt255 := 970, txt_Err_Spn16047_Fmi31_FmiExt255 := 971, txt_Err_Spn16052_Fmi31_FmiExt255 := 972, txt_Err_Spn16057_Fmi31_FmiExt255 := 973, txt_Err_Spn16058_Fmi31_FmiExt255 := 974, txt_Err_Spn16059_Fmi31_FmiExt255 := 975, txt_Err_Spn16060_Fmi31_FmiExt255 := 976, txt_Err_Spn16065_Fmi31_FmiExt255 := 977, txt_Err_Spn16066_Fmi31_FmiExt255 := 978, txt_Err_Spn16067_Fmi31_FmiExt255 := 979, txt_Err_Spn16069_Fmi31_FmiExt255 := 980, txt_Err_Spn16071_Fmi31_FmiExt255 := 981, txt_Err_Spn16072_Fmi31_FmiExt255 := 982, txt_Err_Spn16073_Fmi31_FmiExt255 := 983, txt_Err_Spn16074_Fmi31_FmiExt255 := 984, txt_Err_Spn16075_Fmi31_FmiExt255 := 985, txt_Err_Spn16076_Fmi31_FmiExt255 := 986, txt_Err_Spn16077_Fmi31_FmiExt255 := 987, txt_Err_Spn16078_Fmi31_FmiExt255 := 988, txt_Err_Spn16079_Fmi31_FmiExt255 := 989, txt_Err_Spn16080_Fmi31_FmiExt255 := 990, txt_Err_Spn16081_Fmi31_FmiExt255 := 991, txt_Err_Spn16082_Fmi24_FmiExt255 := 992, txt_Err_Spn16083_Fmi31_FmiExt255 := 993, txt_Err_Spn16084_Fmi31_FmiExt255 := 994, txt_Err_Spn16085_Fmi31_FmiExt255 := 995, txt_Err_Spn16086_Fmi31_FmiExt255 := 996, txt_Err_Spn16087_Fmi31_FmiExt255 := 997, txt_Err_Spn16088_Fmi31_FmiExt255 := 998, txt_Err_Spn16090_Fmi31_FmiExt255 := 999, txt_Err_Spn16099_Fmi31_FmiExt255 := 1000, txt_Err_Spn16100_Fmi31_FmiExt255 := 1001, txt_Err_Spn16101_Fmi31_FmiExt255 := 1002, txt_Err_Spn16122_Fmi31_FmiExt255 := 1003, txt_Err_Spn16123_Fmi31_FmiExt255 := 1004, txt_Err_Spn16124_Fmi31_FmiExt255 := 1005, txt_Err_Spn16125_Fmi31_FmiExt255 := 1006, txt_Err_Spn16128_Fmi31_FmiExt255 := 1007, txt_Err_Spn16129_Fmi31_FmiExt255 := 1008, txt_Err_Spn16130_Fmi31_FmiExt255 := 1009, txt_Err_Spn16131_Fmi31_FmiExt255 := 1010, txt_Err_Spn16134_Fmi31_FmiExt255 := 1011, txt_Err_Spn16135_Fmi31_FmiExt255 := 1012, txt_Err_Spn16136_Fmi31_FmiExt255 := 1013, txt_Err_Spn16137_Fmi31_FmiExt255 := 1014, txt_Err_Spn16138_Fmi31_FmiExt255 := 1015, txt_Err_Spn16139_Fmi31_FmiExt255 := 1016, txt_Err_Spn16140_Fmi31_FmiExt255 := 1017, txt_Err_Spn16141_Fmi31_FmiExt255 := 1018, txt_Err_Spn16142_Fmi31_FmiExt255 := 1019, txt_Err_Spn16143_Fmi31_FmiExt255 := 1020, txt_Err_Spn16144_Fmi31_FmiExt255 := 1021, txt_Err_Spn16148_Fmi31_FmiExt255 := 1022, txt_Err_Spn16152_Fmi31_FmiExt255 := 1023, txt_Err_Spn16153_Fmi31_FmiExt255 := 1024, txt_Err_Spn16154_Fmi31_FmiExt255 := 1025, txt_Err_Spn16155_Fmi31_FmiExt255 := 1026, txt_Err_Spn16157_Fmi31_FmiExt255 := 1027, txt_Err_Spn16158_Fmi31_FmiExt255 := 1028, txt_Err_Spn16159_Fmi31_FmiExt255 := 1029, txt_Err_Spn16161_Fmi31_FmiExt255 := 1030, txt_Err_Spn16162_Fmi31_FmiExt255 := 1031, txt_Err_Spn16163_Fmi31_FmiExt255 := 1032, txt_Err_Spn16164_Fmi31_FmiExt255 := 1033, txt_Err_Spn16166_Fmi31_FmiExt255 := 1034, txt_Err_Spn16178_Fmi31_FmiExt255 := 1035, txt_Err_Spn16182_Fmi31_FmiExt255 := 1036, txt_Err_Spn16183_Fmi31_FmiExt255 := 1037, txt_Err_Spn16184_Fmi31_FmiExt255 := 1038, txt_Err_Spn16186_Fmi31_FmiExt255 := 1039, txt_Err_Spn16192_Fmi31_FmiExt255 := 1040, txt_Err_Spn16193_Fmi31_FmiExt255 := 1041, txt_Err_Spn16194_Fmi31_FmiExt255 := 1042, txt_Err_Spn16196_Fmi31_FmiExt255 := 1043, txt_Err_Spn16205_Fmi31_FmiExt255 := 1044, txt_Err_Spn16213_Fmi31_FmiExt255 := 1045, txt_Err_Spn16214_Fmi31_FmiExt255 := 1046, txt_Err_Spn16215_Fmi31_FmiExt255 := 1047, txt_Err_Spn16239_Fmi31_FmiExt255 := 1048, txt_Err_Spn16240_Fmi31_FmiExt255 := 1049, txt_Err_Spn16241_Fmi31_FmiExt255 := 1050, txt_Err_Spn16244_Fmi31_FmiExt255 := 1051, txt_Err_Spn16245_Fmi31_FmiExt255 := 1052, txt_Err_Spn16246_Fmi31_FmiExt255 := 1053, txt_Err_Spn16251_Fmi31_FmiExt255 := 1054, txt_Err_Spn16252_Fmi31_FmiExt255 := 1055, txt_Err_Spn16253_Fmi31_FmiExt255 := 1056, txt_Err_Spn16255_Fmi31_FmiExt255 := 1057, txt_Err_Spn16262_Fmi31_FmiExt255 := 1058, txt_Err_Spn16264_Fmi31_FmiExt255 := 1059, txt_Err_Spn16265_Fmi31_FmiExt255 := 1060, txt_Err_Spn16266_Fmi31_FmiExt255 := 1061, txt_Err_Spn16267_Fmi31_FmiExt255 := 1062, txt_Err_Spn16272_Fmi31_FmiExt255 := 1063, txt_Err_Spn16276_Fmi31_FmiExt255 := 1064, txt_Err_Spn16277_Fmi31_FmiExt255 := 1065, txt_Err_Spn16278_Fmi31_FmiExt255 := 1066, txt_Err_Spn16280_Fmi31_FmiExt255 := 1067, txt_Err_Spn16296_Fmi31_FmiExt255 := 1068, txt_Err_Spn16297_Fmi31_FmiExt255 := 1069, txt_Err_Spn16298_Fmi31_FmiExt255 := 1070, txt_Err_Spn16300_Fmi31_FmiExt255 := 1071, txt_Err_Spn16302_Fmi31_FmiExt255 := 1072, txt_Err_Spn16303_Fmi31_FmiExt255 := 1073, txt_Err_Spn16304_Fmi31_FmiExt255 := 1074, txt_Err_Spn16305_Fmi31_FmiExt255 := 1075, txt_Err_Spn16306_Fmi31_FmiExt255 := 1076, txt_Err_Spn16307_Fmi31_FmiExt255 := 1077, txt_Err_Spn16308_Fmi24_FmiExt255 := 1078, txt_Err_Spn16309_Fmi31_FmiExt255 := 1079, txt_Err_Spn16310_Fmi31_FmiExt255 := 1080, txt_Err_Spn16311_Fmi24_FmiExt255 := 1081, txt_Err_Spn16312_Fmi31_FmiExt255 := 1082, txt_Err_Spn16313_Fmi31_FmiExt255 := 1083, txt_Err_Spn16314_Fmi31_FmiExt255 := 1084, txt_Err_Spn16315_Fmi31_FmiExt255 := 1085, txt_Err_Spn16316_Fmi31_FmiExt255 := 1086, txt_Err_Spn16317_Fmi31_FmiExt255 := 1087, txt_Err_Spn16318_Fmi31_FmiExt255 := 1088, txt_Err_Spn16319_Fmi31_FmiExt255 := 1089, txt_Err_Spn16320_Fmi31_FmiExt255 := 1090, txt_Err_Spn16321_Fmi31_FmiExt255 := 1091, txt_Err_Spn16322_Fmi31_FmiExt255 := 1092, txt_Err_Spn16323_Fmi31_FmiExt255 := 1093, txt_Err_Spn16324_Fmi31_FmiExt255 := 1094, txt_Err_Spn16325_Fmi31_FmiExt255 := 1095, txt_Err_Spn16326_Fmi31_FmiExt255 := 1096, txt_Err_Spn16327_Fmi31_FmiExt255 := 1097, txt_Err_Spn16328_Fmi24_FmiExt255 := 1098, txt_Err_Spn16329_Fmi24_FmiExt255 := 1099, txt_Err_Spn16330_Fmi31_FmiExt255 := 1100, txt_Err_Spn16331_Fmi31_FmiExt255 := 1101, txt_Err_Spn16336_Fmi31_FmiExt255 := 1102, txt_Err_Spn16337_Fmi31_FmiExt255 := 1103, txt_Err_Spn16341_Fmi31_FmiExt255 := 1104, txt_Err_Spn16342_Fmi31_FmiExt255 := 1105, txt_Err_Spn16344_Fmi31_FmiExt255 := 1106, txt_Err_Spn16345_Fmi31_FmiExt255 := 1107, txt_Err_Spn16347_Fmi31_FmiExt255 := 1108, txt_Err_Spn16354_Fmi31_FmiExt255 := 1109, txt_Err_Spn16360_Fmi31_FmiExt255 := 1110, txt_Err_Spn16361_Fmi31_FmiExt255 := 1111, txt_Err_Spn16363_Fmi31_FmiExt255 := 1112, txt_Err_Spn16439_Fmi31_FmiExt255 := 1113, txt_Err_Spn16457_Fmi31_FmiExt255 := 1114, txt_Err_Spn16465_Fmi31_FmiExt255 := 1115, txt_Err_Spn16470_Fmi31_FmiExt255 := 1116, txt_Err_Spn16472_Fmi31_FmiExt255 := 1117, txt_Err_Spn16473_Fmi31_FmiExt255 := 1118, txt_Err_Spn16475_Fmi31_FmiExt255 := 1119, txt_Err_Spn16476_Fmi31_FmiExt255 := 1120, txt_Err_Spn16477_Fmi31_FmiExt255 := 1121, txt_Err_Spn16479_Fmi31_FmiExt255 := 1122, txt_Err_Spn16505_Fmi31_FmiExt255 := 1123, txt_Err_Spn16510_Fmi31_FmiExt255 := 1124, txt_Err_Spn16514_Fmi31_FmiExt255 := 1125, txt_Err_Spn16515_Fmi31_FmiExt255 := 1126, txt_Err_Spn16516_Fmi31_FmiExt255 := 1127, txt_Err_Spn16517_Fmi31_FmiExt255 := 1128, txt_Err_Spn16518_Fmi31_FmiExt255 := 1129, txt_Err_Spn16519_Fmi31_FmiExt255 := 1130, txt_Err_Spn16520_Fmi31_FmiExt255 := 1131, txt_Err_Spn16521_Fmi31_FmiExt255 := 1132, txt_Err_Spn16522_Fmi31_FmiExt255 := 1133, txt_Err_Spn16523_Fmi31_FmiExt255 := 1134, txt_Err_Spn16524_Fmi31_FmiExt255 := 1135, txt_Err_Spn16525_Fmi31_FmiExt255 := 1136, txt_Err_Spn16526_Fmi31_FmiExt255 := 1137, txt_Err_Spn16527_Fmi31_FmiExt255 := 1138, txt_Err_Spn16528_Fmi31_FmiExt255 := 1139, txt_Err_Spn16529_Fmi31_FmiExt255 := 1140, txt_Err_Spn16530_Fmi31_FmiExt255 := 1141, txt_Err_Spn16531_Fmi31_FmiExt255 := 1142, txt_Err_Spn16532_Fmi31_FmiExt255 := 1143, txt_Err_Spn16533_Fmi31_FmiExt255 := 1144, txt_Err_Spn16534_Fmi31_FmiExt255 := 1145, txt_Err_Spn16535_Fmi31_FmiExt255 := 1146, txt_Err_Spn16536_Fmi31_FmiExt255 := 1147, txt_Err_Spn16537_Fmi31_FmiExt255 := 1148, txt_Err_Spn16538_Fmi31_FmiExt255 := 1149, txt_Err_Spn16539_Fmi31_FmiExt255 := 1150, txt_Err_Spn16540_Fmi31_FmiExt255 := 1151, txt_Err_Spn16541_Fmi31_FmiExt255 := 1152, txt_Err_Spn16542_Fmi31_FmiExt255 := 1153, txt_Err_Spn16543_Fmi31_FmiExt255 := 1154, txt_Err_Spn16544_Fmi31_FmiExt255 := 1155, txt_Err_Spn16545_Fmi31_FmiExt255 := 1156, txt_Err_Spn16547_Fmi31_FmiExt255 := 1157, txt_Err_Spn16548_Fmi31_FmiExt255 := 1158, txt_Err_Spn16549_Fmi31_FmiExt255 := 1159, txt_Err_Spn16551_Fmi31_FmiExt255 := 1160, txt_Err_Spn16552_Fmi31_FmiExt255 := 1161, txt_Err_Spn16553_Fmi31_FmiExt255 := 1162, txt_Err_Spn16554_Fmi31_FmiExt255 := 1163, txt_Err_Spn16555_Fmi31_FmiExt255 := 1164, txt_Err_Spn16556_Fmi31_FmiExt255 := 1165, txt_Err_Spn16557_Fmi31_FmiExt255 := 1166, txt_Err_Spn16558_Fmi31_FmiExt255 := 1167, txt_Err_Spn16559_Fmi31_FmiExt255 := 1168, txt_Err_Spn16560_Fmi31_FmiExt255 := 1169, txt_Err_Spn16561_Fmi31_FmiExt255 := 1170, txt_Err_Spn16562_Fmi31_FmiExt255 := 1171, txt_Err_Spn16563_Fmi31_FmiExt255 := 1172, txt_Err_Spn16564_Fmi31_FmiExt255 := 1173, txt_Err_Spn16565_Fmi31_FmiExt255 := 1174, txt_Err_Spn16566_Fmi31_FmiExt255 := 1175, txt_Err_Spn16577_Fmi31_FmiExt255 := 1176, txt_Err_Spn16578_Fmi31_FmiExt255 := 1177, txt_Err_Spn16583_Fmi31_FmiExt255 := 1178, txt_Err_Spn16588_Fmi31_FmiExt255 := 1179, txt_Err_Spn16589_Fmi31_FmiExt255 := 1180, txt_Err_Spn16590_Fmi31_FmiExt255 := 1181, txt_Err_Spn16591_Fmi31_FmiExt255 := 1182, txt_Err_Spn16592_Fmi31_FmiExt255 := 1183, txt_Err_Spn16593_Fmi31_FmiExt255 := 1184, txt_Err_Spn16595_Fmi31_FmiExt255 := 1185, txt_Err_Spn16596_Fmi31_FmiExt255 := 1186, txt_Err_Spn16597_Fmi31_FmiExt255 := 1187, txt_Err_Spn16598_Fmi31_FmiExt255 := 1188, txt_Err_Spn16599_Fmi31_FmiExt255 := 1189, txt_Err_Spn16611_Fmi31_FmiExt255 := 1190, txt_Err_Spn16612_Fmi31_FmiExt255 := 1191, txt_Err_Spn16613_Fmi31_FmiExt255 := 1192, txt_Err_Spn16614_Fmi31_FmiExt255 := 1193) UINT;
END_TYPE

VAR_GLOBAL CONSTANT  (* ErrDescriptions *)
  gc_ErrTranslation_de_Text0 : WSTRING(40) := " [-]: Ecu0_Safety -  DM_ECU0_INPBOARDNON";
  gc_ErrTranslation_de_Text1 : WSTRING(40) := " [-]: Ecu0_Safety -  DM_ECU0_INPBOARDFAT";
  gc_ErrTranslation_de_Text2 : WSTRING(38) := " [-]: Ecu0_Safety -  DM_ECU0_INPUTPINS";
  gc_ErrTranslation_de_Text3 : WSTRING(67) := " [-]: Ecu0_Safety -  Digital pin error - check ECU hardware and EMI";
  gc_ErrTranslation_de_Text4 : WSTRING(66) := " [-]: Ecu0_Safety -  PWM output error - check ECU hardware and EMI";
  gc_ErrTranslation_de_Text5 : WSTRING(63) := " [-]: Ecu0_Safety -  CPU core error - check source code and EMI";
  gc_ErrTranslation_de_Text6 : WSTRING(33) := " [-]: Ecu0_Safety -  Memory error";
  gc_ErrTranslation_de_Text7 : WSTRING(86) := " [-]: Ecu0_Safety -  Error during watchdog startup - check watchdog timing constraints";
  gc_ErrTranslation_de_Text8 : WSTRING(88) := " [-]: Ecu1_Safety -  Safety switch error - check external shut-off pins and ECU hardware";
  gc_ErrTranslation_de_Text9 : WSTRING(55) := " [-]: Ecu1_Safety -  Application code called safe state";
  gc_ErrTranslation_de_Text10 : WSTRING(29) := " [-]: CAN_BUS0 -  CAN Bus off";
  gc_ErrTranslation_de_Text11 : WSTRING(29) := " [-]: CAN_BUS0 -  CAN warning";
  gc_ErrTranslation_de_Text12 : WSTRING(65) := " [-]: Ecu1_Safety -  Fatal error caused safe state -  replace ECU";
  gc_ErrTranslation_de_Text13 : WSTRING(62) := " [-]: Ecu1_Safety -  BSP error caused safe state - replace ECU";
  gc_ErrTranslation_de_Text14 : WSTRING(29) := " [-]: EcuSil -  Task overload";
  gc_ErrTranslation_de_Text15 : WSTRING(28) := " [-]: EcuSil -  Batttery Low";
  gc_ErrTranslation_de_Text16 : WSTRING(28) := " [-]: EcuSil -  Battery High";
  gc_ErrTranslation_de_Text17 : WSTRING(31) := " [-]: EcuSil -  Temperature Low";
  gc_ErrTranslation_de_Text18 : WSTRING(32) := " [-]: EcuSil -  Temperature High";
  gc_ErrTranslation_de_Text19 : WSTRING(42) := " [-]: SensorSupply -  Sensor Supply S1 Low";
  gc_ErrTranslation_de_Text20 : WSTRING(43) := " [-]: SensorSupply -  Sensor Supply S1 High";
  gc_ErrTranslation_de_Text21 : WSTRING(42) := " [-]: SensorSupply -  Sensor Supply S2 Low";
  gc_ErrTranslation_de_Text22 : WSTRING(43) := " [-]: SensorSupply -  Sensor Supply S2 High";
  gc_ErrTranslation_de_Text23 : WSTRING(42) := " [-]: SensorSupply -  Sensor Supply 5V Low";
  gc_ErrTranslation_de_Text24 : WSTRING(43) := " [-]: SensorSupply -  Sensor Supply 5V High";
  gc_ErrTranslation_de_Text25 : WSTRING(33) := " [-]: ErrList -  List load oneset";
  gc_ErrTranslation_de_Text26 : WSTRING(33) := " [-]: ErrList -  List load defect";
  gc_ErrTranslation_de_Text27 : WSTRING(34) := " [-]: ErrList -  List store defect";
  gc_ErrTranslation_de_Text28 : WSTRING(29) := " [-]: CAN_BUS0 -  CAN Bus off";
  gc_ErrTranslation_de_Text29 : WSTRING(29) := " [-]: CAN_BUS0 -  CAN warning";
  gc_ErrTranslation_de_Text30 : WSTRING(49) := " [-]: CBUS0_HWBUF_SND0 -  HW-Buffer overflow send";
  gc_ErrTranslation_de_Text31 : WSTRING(49) := " [-]: CBUS0_HWBUF_SND0 -  HW-Buffer overflow send";
  gc_ErrTranslation_de_Text32 : WSTRING(49) := " [-]: CBUS0_HWBUF_SND0 -  HW-Buffer overflow send";
  gc_ErrTranslation_de_Text33 : WSTRING(49) := " [-]: CBUS0_HWBUF_SND0 -  HW-Buffer overflow send";
  gc_ErrTranslation_de_Text34 : WSTRING(49) := " [-]: CBUS0_HWBUF_SND0 -  HW-Buffer overflow send";
  gc_ErrTranslation_de_Text35 : WSTRING(49) := " [-]: CBUS0_HWBUF_SND0 -  HW-Buffer overflow send";
  gc_ErrTranslation_de_Text36 : WSTRING(52) := " [-]: CBUS0_HWBUF_RCV0 -  HW-Buffer overflow receive";
  gc_ErrTranslation_de_Text37 : WSTRING(52) := " [-]: CBUS0_HWBUF_RCV1 -  HW-Buffer overflow receive";
  gc_ErrTranslation_de_Text38 : WSTRING(52) := " [-]: CBUS0_HWBUF_RCV2 -  HW-Buffer overflow receive";
  gc_ErrTranslation_de_Text39 : WSTRING(52) := " [-]: CBUS0_HWBUF_RCV3 -  HW-Buffer overflow receive";
  gc_ErrTranslation_de_Text40 : WSTRING(52) := " [-]: CBUS0_HWBUF_RCV4 -  HW-Buffer overflow receive";
  gc_ErrTranslation_de_Text41 : WSTRING(52) := " [-]: CBUS0_HWBUF_RCV5 -  HW-Buffer overflow receive";
  gc_ErrTranslation_de_Text42 : WSTRING(52) := " [-]: CBUS0_HWBUF_RCV6 -  HW-Buffer overflow receive";
  gc_ErrTranslation_de_Text43 : WSTRING(52) := " [-]: CBUS0_HWBUF_RCV7 -  HW-Buffer overflow receive";
  gc_ErrTranslation_de_Text44 : WSTRING(40) := " [-]: Ecu0_Safety -  DM_ECU0_INPBOARDNON";
  gc_ErrTranslation_de_Text45 : WSTRING(40) := " [-]: Ecu0_Safety -  DM_ECU0_INPBOARDFAT";
  gc_ErrTranslation_de_Text46 : WSTRING(38) := " [-]: Ecu0_Safety -  DM_ECU0_INPUTPINS";
  gc_ErrTranslation_de_Text47 : WSTRING(67) := " [-]: Ecu0_Safety -  Digital pin error - check ECU hardware and EMI";
  gc_ErrTranslation_de_Text48 : WSTRING(66) := " [-]: Ecu0_Safety -  PWM output error - check ECU hardware and EMI";
  gc_ErrTranslation_de_Text49 : WSTRING(63) := " [-]: Ecu0_Safety -  CPU core error - check source code and EMI";
  gc_ErrTranslation_de_Text50 : WSTRING(33) := " [-]: Ecu0_Safety -  Memory error";
  gc_ErrTranslation_de_Text51 : WSTRING(86) := " [-]: Ecu0_Safety -  Error during watchdog startup - check watchdog timing constraints";
  gc_ErrTranslation_de_Text52 : WSTRING(88) := " [-]: Ecu1_Safety -  Safety switch error - check external shut-off pins and ECU hardware";
  gc_ErrTranslation_de_Text53 : WSTRING(55) := " [-]: Ecu1_Safety -  Application code called safe state";
  gc_ErrTranslation_de_Text54 : WSTRING(65) := " [-]: Ecu1_Safety -  Fatal error caused safe state -  replace ECU";
  gc_ErrTranslation_de_Text55 : WSTRING(62) := " [-]: Ecu1_Safety -  BSP error caused safe state - replace ECU";
  gc_ErrTranslation_de_Text56 : WSTRING(29) := " [-]: EcuSil -  Task overload";
  gc_ErrTranslation_de_Text57 : WSTRING(28) := " [-]: EcuSil -  Batttery Low";
  gc_ErrTranslation_de_Text58 : WSTRING(28) := " [-]: EcuSil -  Battery High";
  gc_ErrTranslation_de_Text59 : WSTRING(31) := " [-]: EcuSil -  Temperature Low";
  gc_ErrTranslation_de_Text60 : WSTRING(32) := " [-]: EcuSil -  Temperature High";
  gc_ErrTranslation_de_Text61 : WSTRING(42) := " [-]: SensorSupply -  Sensor Supply S1 Low";
  gc_ErrTranslation_de_Text62 : WSTRING(43) := " [-]: SensorSupply -  Sensor Supply S1 High";
  gc_ErrTranslation_de_Text63 : WSTRING(42) := " [-]: SensorSupply -  Sensor Supply S2 Low";
  gc_ErrTranslation_de_Text64 : WSTRING(43) := " [-]: SensorSupply -  Sensor Supply S2 High";
  gc_ErrTranslation_de_Text65 : WSTRING(42) := " [-]: SensorSupply -  Sensor Supply 5V Low";
  gc_ErrTranslation_de_Text66 : WSTRING(43) := " [-]: SensorSupply -  Sensor Supply 5V High";
  gc_ErrTranslation_de_Text67 : WSTRING(33) := " [-]: ErrList -  List load oneset";
  gc_ErrTranslation_de_Text68 : WSTRING(33) := " [-]: ErrList -  List load defect";
  gc_ErrTranslation_de_Text69 : WSTRING(34) := " [-]: ErrList -  List store defect";
  gc_ErrTranslation_de_Text70 : WSTRING(29) := " [-]: CAN_BUS2 -  CAN Bus off";
  gc_ErrTranslation_de_Text71 : WSTRING(29) := " [-]: CAN_BUS2 -  CAN warning";
  gc_ErrTranslation_de_Text72 : WSTRING(49) := " [-]: CBUS2_HWBUF_SND0 -  HW-Buffer overflow send";
  gc_ErrTranslation_de_Text73 : WSTRING(49) := " [-]: CBUS2_HWBUF_SND0 -  HW-Buffer overflow send";
  gc_ErrTranslation_de_Text74 : WSTRING(49) := " [-]: CBUS2_HWBUF_SND0 -  HW-Buffer overflow send";
  gc_ErrTranslation_de_Text75 : WSTRING(49) := " [-]: CBUS2_HWBUF_SND0 -  HW-Buffer overflow send";
  gc_ErrTranslation_de_Text76 : WSTRING(49) := " [-]: CBUS2_HWBUF_SND0 -  HW-Buffer overflow send";
  gc_ErrTranslation_de_Text77 : WSTRING(49) := " [-]: CBUS2_HWBUF_SND0 -  HW-Buffer overflow send";
  gc_ErrTranslation_de_Text78 : WSTRING(52) := " [-]: CBUS2_HWBUF_RCV0 -  HW-Buffer overflow receive";
  gc_ErrTranslation_de_Text79 : WSTRING(52) := " [-]: CBUS2_HWBUF_RCV1 -  HW-Buffer overflow receive";
  gc_ErrTranslation_de_Text80 : WSTRING(52) := " [-]: CBUS2_HWBUF_RCV2 -  HW-Buffer overflow receive";
  gc_ErrTranslation_de_Text81 : WSTRING(52) := " [-]: CBUS2_HWBUF_RCV3 -  HW-Buffer overflow receive";
  gc_ErrTranslation_de_Text82 : WSTRING(52) := " [-]: CBUS2_HWBUF_RCV4 -  HW-Buffer overflow receive";
  gc_ErrTranslation_de_Text83 : WSTRING(52) := " [-]: CBUS2_HWBUF_RCV5 -  HW-Buffer overflow receive";
  gc_ErrTranslation_de_Text84 : WSTRING(52) := " [-]: CBUS2_HWBUF_RCV6 -  HW-Buffer overflow receive";
  gc_ErrTranslation_de_Text85 : WSTRING(52) := " [-]: CBUS2_HWBUF_RCV7 -  HW-Buffer overflow receive";
  gc_ErrTranslation_de_Text86 : WSTRING(0) := "";
  gc_ErrTranslation_de_Text87 : WSTRING(0) := "";
  gc_ErrTranslation_de_Text88 : WSTRING(0) := "";
  gc_ErrTranslation_de_Text89 : WSTRING(0) := "";
  gc_ErrTranslation_de_Text90 : WSTRING(0) := "";
  gc_ErrTranslation_de_Text91 : WSTRING(0) := "";
  gc_ErrTranslation_de_Text92 : WSTRING(0) := "";
  gc_ErrTranslation_de_Text93 : WSTRING(0) := "";
  gc_ErrTranslation_de_Text94 : WSTRING(0) := "";
  gc_ErrTranslation_de_Text95 : WSTRING(0) := "";
  gc_ErrTranslation_de_Text96 : WSTRING(0) := "";
  gc_ErrTranslation_de_Text97 : WSTRING(0) := "";
  gc_ErrTranslation_de_Text98 : WSTRING(0) := "";
  gc_ErrTranslation_de_Text99 : WSTRING(0) := "";
  gc_ErrTranslation_de_Text100 : WSTRING(0) := "";
  gc_ErrTranslation_de_Text101 : WSTRING(0) := "";
  gc_ErrTranslation_de_Text102 : WSTRING(0) := "";
  gc_ErrTranslation_de_Text103 : WSTRING(0) := "";
  gc_ErrTranslation_de_Text104 : WSTRING(29) := " [-]: CAN_BUS3 -  CAN Bus off";
  gc_ErrTranslation_de_Text105 : WSTRING(29) := " [-]: CAN_BUS3 -  CAN warning";
  gc_ErrTranslation_de_Text106 : WSTRING(49) := " [-]: CBUS3_HWBUF_SND0 -  HW-Buffer overflow send";
  gc_ErrTranslation_de_Text107 : WSTRING(49) := " [-]: CBUS3_HWBUF_SND0 -  HW-Buffer overflow send";
  gc_ErrTranslation_de_Text108 : WSTRING(49) := " [-]: CBUS3_HWBUF_SND0 -  HW-Buffer overflow send";
  gc_ErrTranslation_de_Text109 : WSTRING(49) := " [-]: CBUS3_HWBUF_SND0 -  HW-Buffer overflow send";
  gc_ErrTranslation_de_Text110 : WSTRING(49) := " [-]: CBUS3_HWBUF_SND0 -  HW-Buffer overflow send";
  gc_ErrTranslation_de_Text111 : WSTRING(49) := " [-]: CBUS3_HWBUF_SND0 -  HW-Buffer overflow send";
  gc_ErrTranslation_de_Text112 : WSTRING(52) := " [-]: CBUS3_HWBUF_RCV0 -  HW-Buffer overflow receive";
  gc_ErrTranslation_de_Text113 : WSTRING(52) := " [-]: CBUS3_HWBUF_RCV1 -  HW-Buffer overflow receive";
  gc_ErrTranslation_de_Text114 : WSTRING(52) := " [-]: CBUS3_HWBUF_RCV2 -  HW-Buffer overflow receive";
  gc_ErrTranslation_de_Text115 : WSTRING(52) := " [-]: CBUS3_HWBUF_RCV3 -  HW-Buffer overflow receive";
  gc_ErrTranslation_de_Text116 : WSTRING(52) := " [-]: CBUS3_HWBUF_RCV4 -  HW-Buffer overflow receive";
  gc_ErrTranslation_de_Text117 : WSTRING(52) := " [-]: CBUS3_HWBUF_RCV5 -  HW-Buffer overflow receive";
  gc_ErrTranslation_de_Text118 : WSTRING(52) := " [-]: CBUS3_HWBUF_RCV6 -  HW-Buffer overflow receive";
  gc_ErrTranslation_de_Text119 : WSTRING(52) := " [-]: CBUS3_HWBUF_RCV7 -  HW-Buffer overflow receive";
  gc_ErrTranslation_de_Text120 : WSTRING(0) := "";
  gc_ErrTranslation_de_Text121 : WSTRING(0) := "";
  gc_ErrTranslation_de_Text122 : WSTRING(6) := " [-]: ";
  gc_ErrTranslation_de_Text123 : WSTRING(23) := "Message Buffer Overflow";
  gc_ErrTranslation_de_Text124 : WSTRING(29) := " [-]: CAN_BUS2 -  CAN Bus off";
  gc_ErrTranslation_de_Text125 : WSTRING(29) := " [-]: CAN_BUS2 -  CAN warning";
  gc_ErrTranslation_de_Text126 : WSTRING(49) := " [-]: CBUS2_HWBUF_SND0 -  HW-Buffer overflow send";
  gc_ErrTranslation_de_Text127 : WSTRING(49) := " [-]: CBUS2_HWBUF_SND0 -  HW-Buffer overflow send";
  gc_ErrTranslation_de_Text128 : WSTRING(49) := " [-]: CBUS2_HWBUF_SND0 -  HW-Buffer overflow send";
  gc_ErrTranslation_de_Text129 : WSTRING(49) := " [-]: CBUS2_HWBUF_SND0 -  HW-Buffer overflow send";
  gc_ErrTranslation_de_Text130 : WSTRING(49) := " [-]: CBUS2_HWBUF_SND0 -  HW-Buffer overflow send";
  gc_ErrTranslation_de_Text131 : WSTRING(49) := " [-]: CBUS2_HWBUF_SND0 -  HW-Buffer overflow send";
  gc_ErrTranslation_de_Text132 : WSTRING(52) := " [-]: CBUS2_HWBUF_RCV0 -  HW-Buffer overflow receive";
  gc_ErrTranslation_de_Text133 : WSTRING(52) := " [-]: CBUS2_HWBUF_RCV1 -  HW-Buffer overflow receive";
  gc_ErrTranslation_de_Text134 : WSTRING(52) := " [-]: CBUS2_HWBUF_RCV2 -  HW-Buffer overflow receive";
  gc_ErrTranslation_de_Text135 : WSTRING(52) := " [-]: CBUS2_HWBUF_RCV3 -  HW-Buffer overflow receive";
  gc_ErrTranslation_de_Text136 : WSTRING(52) := " [-]: CBUS2_HWBUF_RCV4 -  HW-Buffer overflow receive";
  gc_ErrTranslation_de_Text137 : WSTRING(52) := " [-]: CBUS2_HWBUF_RCV5 -  HW-Buffer overflow receive";
  gc_ErrTranslation_de_Text138 : WSTRING(52) := " [-]: CBUS2_HWBUF_RCV6 -  HW-Buffer overflow receive";
  gc_ErrTranslation_de_Text139 : WSTRING(52) := " [-]: CBUS2_HWBUF_RCV7 -  HW-Buffer overflow receive";
  gc_ErrTranslation_de_Text140 : WSTRING(0) := "";
  gc_ErrTranslation_de_Text141 : WSTRING(0) := "";
  gc_ErrTranslation_de_Text142 : WSTRING(49) := " [-]: CBUS0_HWBUF_SND0 -  HW-Buffer overflow send";
  gc_ErrTranslation_de_Text143 : WSTRING(49) := " [-]: CBUS0_HWBUF_SND0 -  HW-Buffer overflow send";
  gc_ErrTranslation_de_Text144 : WSTRING(49) := " [-]: CBUS0_HWBUF_SND0 -  HW-Buffer overflow send";
  gc_ErrTranslation_de_Text145 : WSTRING(49) := " [-]: CBUS0_HWBUF_SND0 -  HW-Buffer overflow send";
  gc_ErrTranslation_de_Text146 : WSTRING(49) := " [-]: CBUS0_HWBUF_SND0 -  HW-Buffer overflow send";
  gc_ErrTranslation_de_Text147 : WSTRING(49) := " [-]: CBUS0_HWBUF_SND0 -  HW-Buffer overflow send";
  gc_ErrTranslation_de_Text148 : WSTRING(52) := " [-]: CBUS0_HWBUF_RCV0 -  HW-Buffer overflow receive";
  gc_ErrTranslation_de_Text149 : WSTRING(52) := " [-]: CBUS0_HWBUF_RCV1 -  HW-Buffer overflow receive";
  gc_ErrTranslation_de_Text150 : WSTRING(52) := " [-]: CBUS0_HWBUF_RCV2 -  HW-Buffer overflow receive";
  gc_ErrTranslation_de_Text151 : WSTRING(52) := " [-]: CBUS0_HWBUF_RCV3 -  HW-Buffer overflow receive";
  gc_ErrTranslation_de_Text152 : WSTRING(52) := " [-]: CBUS0_HWBUF_RCV4 -  HW-Buffer overflow receive";
  gc_ErrTranslation_de_Text153 : WSTRING(52) := " [-]: CBUS0_HWBUF_RCV5 -  HW-Buffer overflow receive";
  gc_ErrTranslation_de_Text154 : WSTRING(52) := " [-]: CBUS0_HWBUF_RCV6 -  HW-Buffer overflow receive";
  gc_ErrTranslation_de_Text155 : WSTRING(52) := " [-]: CBUS0_HWBUF_RCV7 -  HW-Buffer overflow receive";
  gc_ErrTranslation_de_Text156 : WSTRING(26) := "Time out of cyclic message";
  gc_ErrTranslation_de_Text157 : WSTRING(23) := "Message Buffer Overflow";
  gc_ErrTranslation_de_Text158 : WSTRING(15) := "Invalid Message";
  gc_ErrTranslation_de_Text159 : WSTRING(11) := "Count Fault";
  gc_ErrTranslation_de_Text160 : WSTRING(8) := "Timeslot";
  gc_ErrTranslation_de_Text161 : WSTRING(26) := "Time out of cyclic message";
  gc_ErrTranslation_de_Text162 : WSTRING(23) := "Message Buffer Overflow";
  gc_ErrTranslation_de_Text163 : WSTRING(15) := "Invalid Message";
  gc_ErrTranslation_de_Text164 : WSTRING(11) := "Count Fault";
  gc_ErrTranslation_de_Text165 : WSTRING(8) := "Timeslot";
  gc_ErrTranslation_de_Text166 : WSTRING(26) := "Time out of cyclic message";
  gc_ErrTranslation_de_Text167 : WSTRING(23) := "Message Buffer Overflow";
  gc_ErrTranslation_de_Text168 : WSTRING(15) := "Invalid Message";
  gc_ErrTranslation_de_Text169 : WSTRING(11) := "Count Fault";
  gc_ErrTranslation_de_Text170 : WSTRING(8) := "Timeslot";
  gc_ErrTranslation_de_Text171 : WSTRING(26) := "Time out of cyclic message";
  gc_ErrTranslation_de_Text172 : WSTRING(23) := "Message Buffer Overflow";
  gc_ErrTranslation_de_Text173 : WSTRING(15) := "Invalid Message";
  gc_ErrTranslation_de_Text174 : WSTRING(11) := "Count Fault";
  gc_ErrTranslation_de_Text175 : WSTRING(8) := "Timeslot";
  gc_ErrTranslation_de_Text176 : WSTRING(26) := "Time out of cyclic message";
  gc_ErrTranslation_de_Text177 : WSTRING(23) := "Message Buffer Overflow";
  gc_ErrTranslation_de_Text178 : WSTRING(15) := "Invalid Message";
  gc_ErrTranslation_de_Text179 : WSTRING(11) := "Count Fault";
  gc_ErrTranslation_de_Text180 : WSTRING(29) := " [-]: CAN_BUS1 -  CAN Bus off";
  gc_ErrTranslation_de_Text181 : WSTRING(29) := " [-]: CAN_BUS1 -  CAN warning";
  gc_ErrTranslation_de_Text182 : WSTRING(49) := " [-]: CBUS1_HWBUF_SND0 -  HW-Buffer overflow send";
  gc_ErrTranslation_de_Text183 : WSTRING(49) := " [-]: CBUS1_HWBUF_SND0 -  HW-Buffer overflow send";
  gc_ErrTranslation_de_Text184 : WSTRING(49) := " [-]: CBUS1_HWBUF_SND0 -  HW-Buffer overflow send";
  gc_ErrTranslation_de_Text185 : WSTRING(49) := " [-]: CBUS1_HWBUF_SND0 -  HW-Buffer overflow send";
  gc_ErrTranslation_de_Text186 : WSTRING(49) := " [-]: CBUS1_HWBUF_SND0 -  HW-Buffer overflow send";
  gc_ErrTranslation_de_Text187 : WSTRING(49) := " [-]: CBUS1_HWBUF_SND0 -  HW-Buffer overflow send";
  gc_ErrTranslation_de_Text188 : WSTRING(52) := " [-]: CBUS1_HWBUF_RCV0 -  HW-Buffer overflow receive";
  gc_ErrTranslation_de_Text189 : WSTRING(52) := " [-]: CBUS1_HWBUF_RCV1 -  HW-Buffer overflow receive";
  gc_ErrTranslation_de_Text190 : WSTRING(52) := " [-]: CBUS1_HWBUF_RCV2 -  HW-Buffer overflow receive";
  gc_ErrTranslation_de_Text191 : WSTRING(52) := " [-]: CBUS1_HWBUF_RCV3 -  HW-Buffer overflow receive";
  gc_ErrTranslation_de_Text192 : WSTRING(52) := " [-]: CBUS1_HWBUF_RCV4 -  HW-Buffer overflow receive";
  gc_ErrTranslation_de_Text193 : WSTRING(52) := " [-]: CBUS1_HWBUF_RCV5 -  HW-Buffer overflow receive";
  gc_ErrTranslation_de_Text194 : WSTRING(52) := " [-]: CBUS1_HWBUF_RCV6 -  HW-Buffer overflow receive";
  gc_ErrTranslation_de_Text195 : WSTRING(52) := " [-]: CBUS1_HWBUF_RCV7 -  HW-Buffer overflow receive";
  gc_ErrTranslation_de_Text196 : WSTRING(29) := " [-]: CAN_BUS1 -  CAN Bus off";
  gc_ErrTranslation_de_Text197 : WSTRING(29) := " [-]: CAN_BUS1 -  CAN warning";
  gc_ErrTranslation_de_Text198 : WSTRING(49) := " [-]: CBUS1_HWBUF_SND0 -  HW-Buffer overflow send";
  gc_ErrTranslation_de_Text199 : WSTRING(49) := " [-]: CBUS1_HWBUF_SND0 -  HW-Buffer overflow send";
  gc_ErrTranslation_de_Text200 : WSTRING(49) := " [-]: CBUS1_HWBUF_SND0 -  HW-Buffer overflow send";
  gc_ErrTranslation_de_Text201 : WSTRING(49) := " [-]: CBUS1_HWBUF_SND0 -  HW-Buffer overflow send";
  gc_ErrTranslation_de_Text202 : WSTRING(49) := " [-]: CBUS1_HWBUF_SND0 -  HW-Buffer overflow send";
  gc_ErrTranslation_de_Text203 : WSTRING(49) := " [-]: CBUS1_HWBUF_SND0 -  HW-Buffer overflow send";
  gc_ErrTranslation_de_Text204 : WSTRING(52) := " [-]: CBUS1_HWBUF_RCV0 -  HW-Buffer overflow receive";
  gc_ErrTranslation_de_Text205 : WSTRING(52) := " [-]: CBUS1_HWBUF_RCV1 -  HW-Buffer overflow receive";
  gc_ErrTranslation_de_Text206 : WSTRING(52) := " [-]: CBUS1_HWBUF_RCV2 -  HW-Buffer overflow receive";
  gc_ErrTranslation_de_Text207 : WSTRING(52) := " [-]: CBUS1_HWBUF_RCV3 -  HW-Buffer overflow receive";
  gc_ErrTranslation_de_Text208 : WSTRING(52) := " [-]: CBUS1_HWBUF_RCV4 -  HW-Buffer overflow receive";
  gc_ErrTranslation_de_Text209 : WSTRING(52) := " [-]: CBUS1_HWBUF_RCV5 -  HW-Buffer overflow receive";
  gc_ErrTranslation_de_Text210 : WSTRING(52) := " [-]: CBUS1_HWBUF_RCV6 -  HW-Buffer overflow receive";
  gc_ErrTranslation_de_Text211 : WSTRING(52) := " [-]: CBUS1_HWBUF_RCV7 -  HW-Buffer overflow receive";
  gc_ErrTranslation_de_Text212 : WSTRING(8) := "Timeslot";
  gc_ErrTranslation_de_Text213 : WSTRING(26) := "Time out of cyclic message";
  gc_ErrTranslation_de_Text214 : WSTRING(23) := "Message Buffer Overflow";
  gc_ErrTranslation_de_Text215 : WSTRING(15) := "Invalid Message";
  gc_ErrTranslation_de_Text216 : WSTRING(11) := "Count Fault";
  gc_ErrTranslation_de_Text217 : WSTRING(8) := "Timeslot";
  gc_ErrTranslation_de_Text218 : WSTRING(18) := "DMx protocol error";
  gc_ErrTranslation_de_Text219 : WSTRING(16) := "CAN Snd Overflow";
  gc_ErrTranslation_de_Text220 : WSTRING(18) := "DMx protocol error";
  gc_ErrTranslation_de_Text221 : WSTRING(16) := "CAN Snd Overflow";
  gc_ErrTranslation_de_Text222 : WSTRING(0) := "";
  gc_ErrTranslation_de_Text223 : WSTRING(0) := "";
  gc_ErrTranslation_de_Text224 : WSTRING(0) := "";
  gc_ErrTranslation_de_Text225 : WSTRING(23) := "Message buffer overflow";
  gc_ErrTranslation_de_Text226 : WSTRING(26) := "Time out of cyclic message";
  gc_ErrTranslation_de_Text227 : WSTRING(23) := "Message buffer overflow";
  gc_ErrTranslation_de_Text228 : WSTRING(15) := "Invalid message";
  gc_ErrTranslation_de_Text229 : WSTRING(11) := "Count fault";
  gc_ErrTranslation_de_Text230 : WSTRING(8) := "Timeslot";
  gc_ErrTranslation_de_Text231 : WSTRING(26) := "Time out of cyclic message";
  gc_ErrTranslation_de_Text232 : WSTRING(23) := "Message buffer overflow";
  gc_ErrTranslation_de_Text233 : WSTRING(15) := "Invalid message";
  gc_ErrTranslation_de_Text234 : WSTRING(11) := "Count fault";
  gc_ErrTranslation_de_Text235 : WSTRING(8) := "Timeslot";
  gc_ErrTranslation_de_Text236 : WSTRING(23) := "Message buffer overflow";
  gc_ErrTranslation_de_Text237 : WSTRING(0) := "";
  gc_ErrTranslation_de_Text238 : WSTRING(0) := "";
  gc_ErrTranslation_de_Text239 : WSTRING(0) := "";
  gc_ErrTranslation_de_Text240 : WSTRING(26) := "Time out of cyclic message";
  gc_ErrTranslation_de_Text241 : WSTRING(23) := "Message buffer overflow";
  gc_ErrTranslation_de_Text242 : WSTRING(15) := "Invalid message";
  gc_ErrTranslation_de_Text243 : WSTRING(11) := "Count fault";
  gc_ErrTranslation_de_Text244 : WSTRING(8) := "Timeslot";
  gc_ErrTranslation_de_Text245 : WSTRING(26) := "Time out of cyclic message";
  gc_ErrTranslation_de_Text246 : WSTRING(23) := "Message buffer overflow";
  gc_ErrTranslation_de_Text247 : WSTRING(15) := "Invalid message";
  gc_ErrTranslation_de_Text248 : WSTRING(11) := "Count fault";
  gc_ErrTranslation_de_Text249 : WSTRING(8) := "Timeslot";
  gc_ErrTranslation_de_Text250 : WSTRING(26) := "Time out of cyclic message";
  gc_ErrTranslation_de_Text251 : WSTRING(23) := "Message buffer overflow";
  gc_ErrTranslation_de_Text252 : WSTRING(15) := "Invalid message";
  gc_ErrTranslation_de_Text253 : WSTRING(11) := "Count fault";
  gc_ErrTranslation_de_Text254 : WSTRING(8) := "Timeslot";
  gc_ErrTranslation_de_Text255 : WSTRING(26) := "Time out of cyclic message";
  gc_ErrTranslation_de_Text256 : WSTRING(23) := "Message buffer overflow";
  gc_ErrTranslation_de_Text257 : WSTRING(15) := "Invalid message";
  gc_ErrTranslation_de_Text258 : WSTRING(11) := "Count fault";
  gc_ErrTranslation_de_Text259 : WSTRING(8) := "Timeslot";
  gc_ErrTranslation_de_Text260 : WSTRING(26) := "Time out of cyclic message";
  gc_ErrTranslation_de_Text261 : WSTRING(23) := "Message buffer overflow";
  gc_ErrTranslation_de_Text262 : WSTRING(15) := "Invalid message";
  gc_ErrTranslation_de_Text263 : WSTRING(11) := "Count fault";
  gc_ErrTranslation_de_Text264 : WSTRING(8) := "Timeslot";
  gc_ErrTranslation_de_Text265 : WSTRING(23) := "Message buffer overflow";
  gc_ErrTranslation_de_Text266 : WSTRING(23) := "Message buffer overflow";
  gc_ErrTranslation_de_Text267 : WSTRING(23) := "Message buffer overflow";
  gc_ErrTranslation_de_Text268 : WSTRING(23) := "Message buffer overflow";
  gc_ErrTranslation_de_Text269 : WSTRING(23) := "Message buffer overflow";
  gc_ErrTranslation_de_Text270 : WSTRING(23) := "Message buffer overflow";
  gc_ErrTranslation_de_Text271 : WSTRING(23) := "Message buffer overflow";
  gc_ErrTranslation_de_Text272 : WSTRING(23) := "Message buffer overflow";
  gc_ErrTranslation_de_Text273 : WSTRING(26) := "Time out of cyclic message";
  gc_ErrTranslation_de_Text274 : WSTRING(23) := "Message buffer overflow";
  gc_ErrTranslation_de_Text275 : WSTRING(15) := "Invalid message";
  gc_ErrTranslation_de_Text276 : WSTRING(11) := "Count fault";
  gc_ErrTranslation_de_Text277 : WSTRING(8) := "Timeslot";
  gc_ErrTranslation_de_Text278 : WSTRING(23) := "Message buffer overflow";
  gc_ErrTranslation_de_Text279 : WSTRING(26) := "Time out of cyclic message";
  gc_ErrTranslation_de_Text280 : WSTRING(23) := "Message buffer overflow";
  gc_ErrTranslation_de_Text281 : WSTRING(15) := "Invalid message";
  gc_ErrTranslation_de_Text282 : WSTRING(11) := "Count fault";
  gc_ErrTranslation_de_Text283 : WSTRING(8) := "Timeslot";
  gc_ErrTranslation_de_Text284 : WSTRING(23) := "Message buffer overflow";
  gc_ErrTranslation_de_Text285 : WSTRING(26) := "Time out of cyclic message";
  gc_ErrTranslation_de_Text286 : WSTRING(23) := "Message buffer overflow";
  gc_ErrTranslation_de_Text287 : WSTRING(15) := "Invalid message";
  gc_ErrTranslation_de_Text288 : WSTRING(11) := "Count fault";
  gc_ErrTranslation_de_Text289 : WSTRING(8) := "Timeslot";
  gc_ErrTranslation_de_Text290 : WSTRING(26) := "Time out of cyclic message";
  gc_ErrTranslation_de_Text291 : WSTRING(23) := "Message buffer overflow";
  gc_ErrTranslation_de_Text292 : WSTRING(15) := "Invalid message";
  gc_ErrTranslation_de_Text293 : WSTRING(11) := "Count fault";
  gc_ErrTranslation_de_Text294 : WSTRING(8) := "Timeslot";
  gc_ErrTranslation_de_Text295 : WSTRING(26) := "Time out of cyclic message";
  gc_ErrTranslation_de_Text296 : WSTRING(23) := "Message buffer overflow";
  gc_ErrTranslation_de_Text297 : WSTRING(15) := "Invalid message";
  gc_ErrTranslation_de_Text298 : WSTRING(11) := "Count fault";
  gc_ErrTranslation_de_Text299 : WSTRING(8) := "Timeslot";
  gc_ErrTranslation_de_Text300 : WSTRING(23) := "Message buffer overflow";
  gc_ErrTranslation_de_Text301 : WSTRING(23) := "Message buffer overflow";
  gc_ErrTranslation_de_Text302 : WSTRING(81) := " [PIN_103 ]: PressureBlockOscillationSensor -  Master input signal short to power";
  gc_ErrTranslation_de_Text303 : WSTRING(82) := " [PIN_103 ]: PressureBlockOscillationSensor -  Master input signal short to ground";
  gc_ErrTranslation_de_Text304 : WSTRING(82) := " [PIN_103 ]: PressureBlockOscillationSensor -  Parameter of input char NOT monoton";
  gc_ErrTranslation_de_Text305 : WSTRING(69) := " [PIN_103 ]: PressureBlockOscillationSensor -  Unknown internal error";
  gc_ErrTranslation_de_Text306 : WSTRING(70) := " [PIN_127 ]: PressureBrakeSensor -  Master input signal short to power";
  gc_ErrTranslation_de_Text307 : WSTRING(71) := " [PIN_127 ]: PressureBrakeSensor -  Master input signal short to ground";
  gc_ErrTranslation_de_Text308 : WSTRING(71) := " [PIN_127 ]: PressureBrakeSensor -  Parameter of input char NOT monoton";
  gc_ErrTranslation_de_Text309 : WSTRING(58) := " [PIN_127 ]: PressureBrakeSensor -  Unknown internal error";
  gc_ErrTranslation_de_Text310 : WSTRING(78) := " [PIN_103 ]: Transmission1PressureSensor -  Master input signal short to power";
  gc_ErrTranslation_de_Text311 : WSTRING(79) := " [PIN_103 ]: Transmission1PressureSensor -  Master input signal short to ground";
  gc_ErrTranslation_de_Text312 : WSTRING(79) := " [PIN_103 ]: Transmission1PressureSensor -  Parameter of input char NOT monoton";
  gc_ErrTranslation_de_Text313 : WSTRING(66) := " [PIN_103 ]: Transmission1PressureSensor -  Unknown internal error";
  gc_ErrTranslation_de_Text314 : WSTRING(27) := " [-]: SpecificErrorC0_5 -  ";
  gc_ErrTranslation_de_Text315 : WSTRING(27) := " [-]: SpecificErrorC0_5 -  ";
  gc_ErrTranslation_de_Text316 : WSTRING(77) := " [-]: SpecificErrorC0_5 -  Check pressure when bypass is pilot detected by C1";
  gc_ErrTranslation_de_Text317 : WSTRING(27) := " [-]: SpecificErrorC0_5 -  ";
  gc_ErrTranslation_de_Text318 : WSTRING(38) := " [-]: SpecificErrorC0_5 -  Error bit 4";
  gc_ErrTranslation_de_Text319 : WSTRING(38) := " [-]: SpecificErrorC0_5 -  Error bit 5";
  gc_ErrTranslation_de_Text320 : WSTRING(38) := " [-]: SpecificErrorC0_5 -  Error bit 6";
  gc_ErrTranslation_de_Text321 : WSTRING(9) := "DMC error";
  gc_ErrTranslation_de_Text322 : WSTRING(65) := " [PIN_115 ]: OscillantAxleSpeedSensor -  Input is short to Ground";
  gc_ErrTranslation_de_Text323 : WSTRING(64) := " [PIN_115 ]: OscillantAxleSpeedSensor -  Input is short to Power";
  gc_ErrTranslation_de_Text324 : WSTRING(56) := " [PIN_115 ]: OscillantAxleSpeedSensor -  Wrong Parameter";
  gc_ErrTranslation_de_Text325 : WSTRING(54) := " [PIN_115 ]: OscillantAxleSpeedSensor -  Unknown Error";
  gc_ErrTranslation_de_Text326 : WSTRING(60) := " [PIN_116 ]: FixeAxleSpeedSensor -  Input is short to Ground";
  gc_ErrTranslation_de_Text327 : WSTRING(59) := " [PIN_116 ]: FixeAxleSpeedSensor -  Input is short to Power";
  gc_ErrTranslation_de_Text328 : WSTRING(51) := " [PIN_116 ]: FixeAxleSpeedSensor -  Wrong Parameter";
  gc_ErrTranslation_de_Text329 : WSTRING(49) := " [PIN_116 ]: FixeAxleSpeedSensor -  Unknown Error";
  gc_ErrTranslation_de_Text330 : WSTRING(77) := " [PIN_153 ]: EvDeflectorTransmission -  HS OpenLoad / Short To Power external";
  gc_ErrTranslation_de_Text331 : WSTRING(66) := " [PIN_153 ]: EvDeflectorTransmission -  HS Short To Power internal";
  gc_ErrTranslation_de_Text332 : WSTRING(58) := " [PIN_153 ]: EvDeflectorTransmission -  HS Short To Ground";
  gc_ErrTranslation_de_Text333 : WSTRING(61) := " [PIN_153 ]: EvDeflectorTransmission -  Internal Driver Error";
  gc_ErrTranslation_de_Text334 : WSTRING(71) := " [PIN_190 ]: EvUpMeasuringMast -  HS OpenLoad / Short To Power external";
  gc_ErrTranslation_de_Text335 : WSTRING(60) := " [PIN_190 ]: EvUpMeasuringMast -  HS Short To Power internal";
  gc_ErrTranslation_de_Text336 : WSTRING(52) := " [PIN_190 ]: EvUpMeasuringMast -  HS Short To Ground";
  gc_ErrTranslation_de_Text337 : WSTRING(55) := " [PIN_190 ]: EvUpMeasuringMast -  Internal Driver Error";
  gc_ErrTranslation_de_Text338 : WSTRING(73) := " [PIN_166 ]: EvDownMeasuringMast -  HS OpenLoad / Short To Power external";
  gc_ErrTranslation_de_Text339 : WSTRING(62) := " [PIN_166 ]: EvDownMeasuringMast -  HS Short To Power internal";
  gc_ErrTranslation_de_Text340 : WSTRING(54) := " [PIN_166 ]: EvDownMeasuringMast -  HS Short To Ground";
  gc_ErrTranslation_de_Text341 : WSTRING(57) := " [PIN_166 ]: EvDownMeasuringMast -  Internal Driver Error";
  gc_ErrTranslation_de_Text342 : WSTRING(73) := " [PIN_195 ]: EvServiceBrakeTrack -  HS OpenLoad / Short To Power external";
  gc_ErrTranslation_de_Text343 : WSTRING(62) := " [PIN_195 ]: EvServiceBrakeTrack -  HS Short To Power internal";
  gc_ErrTranslation_de_Text344 : WSTRING(54) := " [PIN_195 ]: EvServiceBrakeTrack -  HS Short To Ground";
  gc_ErrTranslation_de_Text345 : WSTRING(57) := " [PIN_195 ]: EvServiceBrakeTrack -  Internal Driver Error";
  gc_ErrTranslation_de_Text346 : WSTRING(70) := " [PIN_171 ]: EvPowerReduction -  HS OpenLoad / Short To Power external";
  gc_ErrTranslation_de_Text347 : WSTRING(59) := " [PIN_171 ]: EvPowerReduction -  HS Short To Power internal";
  gc_ErrTranslation_de_Text348 : WSTRING(51) := " [PIN_171 ]: EvPowerReduction -  HS Short To Ground";
  gc_ErrTranslation_de_Text349 : WSTRING(54) := " [PIN_171 ]: EvPowerReduction -  Internal Driver Error";
  gc_ErrTranslation_de_Text350 : WSTRING(78) := " [PIN_127 ]: Transmission2PressureSensor -  Master input signal short to power";
  gc_ErrTranslation_de_Text351 : WSTRING(79) := " [PIN_127 ]: Transmission2PressureSensor -  Master input signal short to ground";
  gc_ErrTranslation_de_Text352 : WSTRING(79) := " [PIN_127 ]: Transmission2PressureSensor -  Parameter of input char NOT monoton";
  gc_ErrTranslation_de_Text353 : WSTRING(66) := " [PIN_127 ]: Transmission2PressureSensor -  Unknown internal error";
  gc_ErrTranslation_de_Text354 : WSTRING(75) := " [PIN_131 PIN_122 ]: DownOscillantAxle -  Logical Error between pin 0 and 1";
  gc_ErrTranslation_de_Text355 : WSTRING(60) := " [PIN_131 PIN_122 ]: DownOscillantAxle -  Vin0 < u16VolLoMin";
  gc_ErrTranslation_de_Text356 : WSTRING(60) := " [PIN_131 PIN_122 ]: DownOscillantAxle -  Vin0 > u16VolHiMax";
  gc_ErrTranslation_de_Text357 : WSTRING(74) := " [PIN_131 PIN_122 ]: DownOscillantAxle -  u16VolLoMax < Vin0 < u16VolHiMin";
  gc_ErrTranslation_de_Text358 : WSTRING(73) := " [PIN_160 ]: SupplyRadioReceiver -  HS OpenLoad / Short To Power external";
  gc_ErrTranslation_de_Text359 : WSTRING(62) := " [PIN_160 ]: SupplyRadioReceiver -  HS Short To Power internal";
  gc_ErrTranslation_de_Text360 : WSTRING(54) := " [PIN_160 ]: SupplyRadioReceiver -  HS Short To Ground";
  gc_ErrTranslation_de_Text361 : WSTRING(57) := " [PIN_160 ]: SupplyRadioReceiver -  Internal Driver Error";
  gc_ErrTranslation_de_Text362 : WSTRING(77) := " [PIN_184 ]: BuzzerLynxMovingMachine -  HS OpenLoad / Short To Power external";
  gc_ErrTranslation_de_Text363 : WSTRING(66) := " [PIN_184 ]: BuzzerLynxMovingMachine -  HS Short To Power internal";
  gc_ErrTranslation_de_Text364 : WSTRING(58) := " [PIN_184 ]: BuzzerLynxMovingMachine -  HS Short To Ground";
  gc_ErrTranslation_de_Text365 : WSTRING(61) := " [PIN_184 ]: BuzzerLynxMovingMachine -  Internal Driver Error";
  gc_ErrTranslation_de_Text366 : WSTRING(80) := " [PIN_104 ]: TemperatureTransmissionSensor -  Master input signal short to power";
  gc_ErrTranslation_de_Text367 : WSTRING(81) := " [PIN_104 ]: TemperatureTransmissionSensor -  Master input signal short to ground";
  gc_ErrTranslation_de_Text368 : WSTRING(81) := " [PIN_104 ]: TemperatureTransmissionSensor -  Parameter of input char NOT monoton";
  gc_ErrTranslation_de_Text369 : WSTRING(68) := " [PIN_104 ]: TemperatureTransmissionSensor -  Unknown internal error";
  gc_ErrTranslation_de_Text370 : WSTRING(66) := " [PIN_150 ]: CoolingRelay -  HS OpenLoad / Short To Power external";
  gc_ErrTranslation_de_Text371 : WSTRING(55) := " [PIN_150 ]: CoolingRelay -  HS Short To Power internal";
  gc_ErrTranslation_de_Text372 : WSTRING(47) := " [PIN_150 ]: CoolingRelay -  HS Short To Ground";
  gc_ErrTranslation_de_Text373 : WSTRING(50) := " [PIN_150 ]: CoolingRelay -  Internal Driver Error";
  gc_ErrTranslation_de_Text374 : WSTRING(67) := " [PIN_173 ]: WhiteLightAVD -  HS OpenLoad / Short To Power external";
  gc_ErrTranslation_de_Text375 : WSTRING(56) := " [PIN_173 ]: WhiteLightAVD -  HS Short To Power internal";
  gc_ErrTranslation_de_Text376 : WSTRING(48) := " [PIN_173 ]: WhiteLightAVD -  HS Short To Ground";
  gc_ErrTranslation_de_Text377 : WSTRING(51) := " [PIN_173 ]: WhiteLightAVD -  Internal Driver Error";
  gc_ErrTranslation_de_Text378 : WSTRING(65) := " [PIN_152 ]: RedLightAVG -  HS OpenLoad / Short To Power external";
  gc_ErrTranslation_de_Text379 : WSTRING(54) := " [PIN_152 ]: RedLightAVG -  HS Short To Power internal";
  gc_ErrTranslation_de_Text380 : WSTRING(46) := " [PIN_152 ]: RedLightAVG -  HS Short To Ground";
  gc_ErrTranslation_de_Text381 : WSTRING(49) := " [PIN_152 ]: RedLightAVG -  Internal Driver Error";
  gc_ErrTranslation_de_Text382 : WSTRING(65) := " [PIN_176 ]: RedLightAVD -  HS OpenLoad / Short To Power external";
  gc_ErrTranslation_de_Text383 : WSTRING(54) := " [PIN_176 ]: RedLightAVD -  HS Short To Power internal";
  gc_ErrTranslation_de_Text384 : WSTRING(46) := " [PIN_176 ]: RedLightAVD -  HS Short To Ground";
  gc_ErrTranslation_de_Text385 : WSTRING(49) := " [PIN_176 ]: RedLightAVD -  Internal Driver Error";
  gc_ErrTranslation_de_Text386 : WSTRING(67) := " [PIN_155 ]: WhiteLightARG -  HS OpenLoad / Short To Power external";
  gc_ErrTranslation_de_Text387 : WSTRING(56) := " [PIN_155 ]: WhiteLightARG -  HS Short To Power internal";
  gc_ErrTranslation_de_Text388 : WSTRING(48) := " [PIN_155 ]: WhiteLightARG -  HS Short To Ground";
  gc_ErrTranslation_de_Text389 : WSTRING(51) := " [PIN_155 ]: WhiteLightARG -  Internal Driver Error";
  gc_ErrTranslation_de_Text390 : WSTRING(67) := " [PIN_179 ]: WhiteLightARD -  HS OpenLoad / Short To Power external";
  gc_ErrTranslation_de_Text391 : WSTRING(56) := " [PIN_179 ]: WhiteLightARD -  HS Short To Power internal";
  gc_ErrTranslation_de_Text392 : WSTRING(48) := " [PIN_179 ]: WhiteLightARD -  HS Short To Ground";
  gc_ErrTranslation_de_Text393 : WSTRING(51) := " [PIN_179 ]: WhiteLightARD -  Internal Driver Error";
  gc_ErrTranslation_de_Text394 : WSTRING(65) := " [PIN_158 ]: RedLightARG -  HS OpenLoad / Short To Power external";
  gc_ErrTranslation_de_Text395 : WSTRING(54) := " [PIN_158 ]: RedLightARG -  HS Short To Power internal";
  gc_ErrTranslation_de_Text396 : WSTRING(46) := " [PIN_158 ]: RedLightARG -  HS Short To Ground";
  gc_ErrTranslation_de_Text397 : WSTRING(49) := " [PIN_158 ]: RedLightARG -  Internal Driver Error";
  gc_ErrTranslation_de_Text398 : WSTRING(65) := " [PIN_182 ]: RedLightARD -  HS OpenLoad / Short To Power external";
  gc_ErrTranslation_de_Text399 : WSTRING(54) := " [PIN_182 ]: RedLightARD -  HS Short To Power internal";
  gc_ErrTranslation_de_Text400 : WSTRING(46) := " [PIN_182 ]: RedLightARD -  HS Short To Ground";
  gc_ErrTranslation_de_Text401 : WSTRING(49) := " [PIN_182 ]: RedLightARD -  Internal Driver Error";
  gc_ErrTranslation_de_Text402 : WSTRING(73) := " [PIN_164 ]: SupplyPvgRightTrack -  HS OpenLoad / Short To Power external";
  gc_ErrTranslation_de_Text403 : WSTRING(62) := " [PIN_164 ]: SupplyPvgRightTrack -  HS Short To Power internal";
  gc_ErrTranslation_de_Text404 : WSTRING(54) := " [PIN_164 ]: SupplyPvgRightTrack -  HS Short To Ground";
  gc_ErrTranslation_de_Text405 : WSTRING(57) := " [PIN_164 ]: SupplyPvgRightTrack -  Internal Driver Error";
  gc_ErrTranslation_de_Text406 : WSTRING(60) := " [PIN_131 PIN_122 ]: DownOscillantAxle -  Vin1 < u16VolLoMin";
  gc_ErrTranslation_de_Text407 : WSTRING(60) := " [PIN_131 PIN_122 ]: DownOscillantAxle -  Vin1 > u16VolHiMax";
  gc_ErrTranslation_de_Text408 : WSTRING(74) := " [PIN_131 PIN_122 ]: DownOscillantAxle -  u16VolLoMax < Vin1 < u16VolHiMin";
  gc_ErrTranslation_de_Text409 : WSTRING(56) := " [-]: SpecificErrorC1_2 -  Coherence pilotage PVG Ev Tor";
  gc_ErrTranslation_de_Text410 : WSTRING(59) := " [-]: SpecificErrorC1_2 -  Coherence pilotage PVG telescope";
  gc_ErrTranslation_de_Text411 : WSTRING(52) := "An input signal is too low / Short circuit to ground";
  gc_ErrTranslation_de_Text412 : WSTRING(52) := "An input signal is too high / Short circuit to power";
  gc_ErrTranslation_de_Text413 : WSTRING(37) := "An input signal is out of valid range";
  gc_ErrTranslation_de_Text414 : WSTRING(39) := "Warning: a block has limited parameters";
  gc_ErrTranslation_de_Text415 : WSTRING(23) := "An initialization error";
  gc_ErrTranslation_de_Text416 : WSTRING(52) := "An input signal is too low / Short circuit to ground";
  gc_ErrTranslation_de_Text417 : WSTRING(84) := " [PIN_132 ]: UpOscillantAxle -  An input signal is too low / Short circuit to ground";
  gc_ErrTranslation_de_Text418 : WSTRING(84) := " [PIN_132 ]: UpOscillantAxle -  An input signal is too high / Short circuit to power";
  gc_ErrTranslation_de_Text419 : WSTRING(69) := " [PIN_132 ]: UpOscillantAxle -  An input signal is out of valid range";
  gc_ErrTranslation_de_Text420 : WSTRING(71) := " [PIN_132 ]: UpOscillantAxle -  Warning: a block has limited parameters";
  gc_ErrTranslation_de_Text421 : WSTRING(55) := " [PIN_132 ]: UpOscillantAxle -  An initialization error";
  gc_ErrTranslation_de_Text422 : WSTRING(79) := " [PIN_109 ]: UpFixeAxle -  An input signal is too low / Short circuit to ground";
  gc_ErrTranslation_de_Text423 : WSTRING(79) := " [PIN_109 ]: UpFixeAxle -  An input signal is too high / Short circuit to power";
  gc_ErrTranslation_de_Text424 : WSTRING(64) := " [PIN_109 ]: UpFixeAxle -  An input signal is out of valid range";
  gc_ErrTranslation_de_Text425 : WSTRING(66) := " [PIN_109 ]: UpFixeAxle -  Warning: a block has limited parameters";
  gc_ErrTranslation_de_Text426 : WSTRING(50) := " [PIN_109 ]: UpFixeAxle -  An initialization error";
  gc_ErrTranslation_de_Text427 : WSTRING(73) := " [PIN_252 ]: PvgLeftTrackLowside -  HS OpenLoad / Short To Power external";
  gc_ErrTranslation_de_Text428 : WSTRING(62) := " [PIN_252 ]: PvgLeftTrackLowside -  HS Short To Power internal";
  gc_ErrTranslation_de_Text429 : WSTRING(54) := " [PIN_252 ]: PvgLeftTrackLowside -  HS Short To Ground";
  gc_ErrTranslation_de_Text430 : WSTRING(57) := " [PIN_252 ]: PvgLeftTrackLowside -  Internal Driver Error";
  gc_ErrTranslation_de_Text431 : WSTRING(27) := " [-]: SpecificErrorC1_2 -  ";
  gc_ErrTranslation_de_Text432 : WSTRING(27) := " [-]: SpecificErrorC1_2 -  ";
  gc_ErrTranslation_de_Text433 : WSTRING(27) := " [-]: SpecificErrorC1_2 -  ";
  gc_ErrTranslation_de_Text434 : WSTRING(69) := " [-]: SpecificErrorC1_2 -  Inconsistency Nc No logical frame rotation";
  gc_ErrTranslation_de_Text435 : WSTRING(27) := " [-]: SpecificErrorC1_2 -  ";
  gc_ErrTranslation_de_Text436 : WSTRING(27) := " [-]: SpecificErrorC1_2 -  ";
  gc_ErrTranslation_de_Text437 : WSTRING(85) := " [PIN_111 ]: FaultPvgDeltaArm -  An input signal is too low / Short circuit to ground";
  gc_ErrTranslation_de_Text438 : WSTRING(85) := " [PIN_111 ]: FaultPvgDeltaArm -  An input signal is too high / Short circuit to power";
  gc_ErrTranslation_de_Text439 : WSTRING(70) := " [PIN_111 ]: FaultPvgDeltaArm -  An input signal is out of valid range";
  gc_ErrTranslation_de_Text440 : WSTRING(72) := " [PIN_111 ]: FaultPvgDeltaArm -  Warning: a block has limited parameters";
  gc_ErrTranslation_de_Text441 : WSTRING(56) := " [PIN_111 ]: FaultPvgDeltaArm -  An initialization error";
  gc_ErrTranslation_de_Text442 : WSTRING(85) := " [PIN_135 ]: FaultPvgArrowArm -  An input signal is too low / Short circuit to ground";
  gc_ErrTranslation_de_Text443 : WSTRING(85) := " [PIN_135 ]: FaultPvgArrowArm -  An input signal is too high / Short circuit to power";
  gc_ErrTranslation_de_Text444 : WSTRING(70) := " [PIN_135 ]: FaultPvgArrowArm -  An input signal is out of valid range";
  gc_ErrTranslation_de_Text445 : WSTRING(72) := " [PIN_135 ]: FaultPvgArrowArm -  Warning: a block has limited parameters";
  gc_ErrTranslation_de_Text446 : WSTRING(56) := " [PIN_135 ]: FaultPvgArrowArm -  An initialization error";
  gc_ErrTranslation_de_Text447 : WSTRING(89) := " [PIN_112 ]: FaultPvgTelescopeArm -  An input signal is too low / Short circuit to ground";
  gc_ErrTranslation_de_Text448 : WSTRING(89) := " [PIN_112 ]: FaultPvgTelescopeArm -  An input signal is too high / Short circuit to power";
  gc_ErrTranslation_de_Text449 : WSTRING(74) := " [PIN_112 ]: FaultPvgTelescopeArm -  An input signal is out of valid range";
  gc_ErrTranslation_de_Text450 : WSTRING(76) := " [PIN_112 ]: FaultPvgTelescopeArm -  Warning: a block has limited parameters";
  gc_ErrTranslation_de_Text451 : WSTRING(60) := " [PIN_112 ]: FaultPvgTelescopeArm -  An initialization error";
  gc_ErrTranslation_de_Text452 : WSTRING(85) := " [PIN_136 ]: FaultPvgEvProTOR -  An input signal is too low / Short circuit to ground";
  gc_ErrTranslation_de_Text453 : WSTRING(85) := " [PIN_136 ]: FaultPvgEvProTOR -  An input signal is too high / Short circuit to power";
  gc_ErrTranslation_de_Text454 : WSTRING(70) := " [PIN_136 ]: FaultPvgEvProTOR -  An input signal is out of valid range";
  gc_ErrTranslation_de_Text455 : WSTRING(72) := " [PIN_136 ]: FaultPvgEvProTOR -  Warning: a block has limited parameters";
  gc_ErrTranslation_de_Text456 : WSTRING(61) := " [PIN_161 ]: PvgLeftTrack -  Short to Power has been detected";
  gc_ErrTranslation_de_Text457 : WSTRING(62) := " [PIN_161 ]: PvgLeftTrack -  Short to Ground has been detected";
  gc_ErrTranslation_de_Text458 : WSTRING(44) := " [PIN_161 ]: PvgLeftTrack -  Wrong Parameter";
  gc_ErrTranslation_de_Text459 : WSTRING(42) := " [PIN_161 ]: PvgLeftTrack -  Unknown error";
  gc_ErrTranslation_de_Text460 : WSTRING(62) := " [PIN_185 ]: PvgRightTrack -  Short to Power has been detected";
  gc_ErrTranslation_de_Text461 : WSTRING(63) := " [PIN_185 ]: PvgRightTrack -  Short to Ground has been detected";
  gc_ErrTranslation_de_Text462 : WSTRING(45) := " [PIN_185 ]: PvgRightTrack -  Wrong Parameter";
  gc_ErrTranslation_de_Text463 : WSTRING(43) := " [PIN_185 ]: PvgRightTrack -  Unknown error";
  gc_ErrTranslation_de_Text464 : WSTRING(56) := " [PIN_136 ]: FaultPvgEvProTOR -  An initialization error";
  gc_ErrTranslation_de_Text465 : WSTRING(32) := "Short to Power has been detected";
  gc_ErrTranslation_de_Text466 : WSTRING(33) := "Short to Ground has been detected";
  gc_ErrTranslation_de_Text467 : WSTRING(15) := "Wrong Parameter";
  gc_ErrTranslation_de_Text468 : WSTRING(13) := "Unknown error";
  gc_ErrTranslation_de_Text469 : WSTRING(37) := "HS OpenLoad / Short To Power external";
  gc_ErrTranslation_de_Text470 : WSTRING(26) := "HS Short To Power internal";
  gc_ErrTranslation_de_Text471 : WSTRING(18) := "HS Short To Ground";
  gc_ErrTranslation_de_Text472 : WSTRING(21) := "Internal Driver Error";
  gc_ErrTranslation_de_Text473 : WSTRING(37) := "HS OpenLoad / Short To Power external";
  gc_ErrTranslation_de_Text474 : WSTRING(26) := "HS Short To Power internal";
  gc_ErrTranslation_de_Text475 : WSTRING(71) := " [PIN_130 ]: BypassPressureSensor -  Master input signal short to power";
  gc_ErrTranslation_de_Text476 : WSTRING(72) := " [PIN_130 ]: BypassPressureSensor -  Master input signal short to ground";
  gc_ErrTranslation_de_Text477 : WSTRING(72) := " [PIN_130 ]: BypassPressureSensor -  Parameter of input char NOT monoton";
  gc_ErrTranslation_de_Text478 : WSTRING(59) := " [PIN_130 ]: BypassPressureSensor -  Unknown internal error";
  gc_ErrTranslation_de_Text479 : WSTRING(70) := " [PIN_108 PIN_146 ]: DownFixeAxle -  Logical Error between pin 0 and 1";
  gc_ErrTranslation_de_Text480 : WSTRING(55) := " [PIN_108 PIN_146 ]: DownFixeAxle -  Vin0 < u16VolLoMin";
  gc_ErrTranslation_de_Text481 : WSTRING(55) := " [PIN_108 PIN_146 ]: DownFixeAxle -  Vin0 > u16VolHiMax";
  gc_ErrTranslation_de_Text482 : WSTRING(69) := " [PIN_108 PIN_146 ]: DownFixeAxle -  u16VolLoMax < Vin0 < u16VolHiMin";
  gc_ErrTranslation_de_Text483 : WSTRING(55) := " [PIN_108 PIN_146 ]: DownFixeAxle -  Vin1 < u16VolLoMin";
  gc_ErrTranslation_de_Text484 : WSTRING(55) := " [PIN_108 PIN_146 ]: DownFixeAxle -  Vin1 > u16VolHiMax";
  gc_ErrTranslation_de_Text485 : WSTRING(69) := " [PIN_108 PIN_146 ]: DownFixeAxle -  u16VolLoMax < Vin1 < u16VolHiMin";
  gc_ErrTranslation_de_Text486 : WSTRING(52) := "An input signal is too high / Short circuit to power";
  gc_ErrTranslation_de_Text487 : WSTRING(37) := "An input signal is out of valid range";
  gc_ErrTranslation_de_Text488 : WSTRING(52) := " [PIN_106 ]: GasGauge -  Input signal short to power";
  gc_ErrTranslation_de_Text489 : WSTRING(53) := " [PIN_106 ]: GasGauge -  Input signal short to ground";
  gc_ErrTranslation_de_Text490 : WSTRING(45) := " [PIN_106 ]: GasGauge -  Internal Block error";
  gc_ErrTranslation_de_Text491 : WSTRING(39) := "Warning: a block has limited parameters";
  gc_ErrTranslation_de_Text492 : WSTRING(23) := "An initialization error";
  gc_ErrTranslation_de_Text493 : WSTRING(49) := "Openload detected on red light ARD output of 48xs";
  gc_ErrTranslation_de_Text494 : WSTRING(33) := "Fault on thermic or electric pump";
  gc_ErrTranslation_de_Text495 : WSTRING(11) := "Error bit 2";
  gc_ErrTranslation_de_Text496 : WSTRING(11) := "Error bit 3";
  gc_ErrTranslation_de_Text497 : WSTRING(11) := "Error bit 4";
  gc_ErrTranslation_de_Text498 : WSTRING(11) := "Error bit 5";
  gc_ErrTranslation_de_Text499 : WSTRING(74) := " [PIN_239 ]: PvgRightTrackLowside -  HS OpenLoad / Short To Power external";
  gc_ErrTranslation_de_Text500 : WSTRING(63) := " [PIN_239 ]: PvgRightTrackLowside -  HS Short To Power internal";
  gc_ErrTranslation_de_Text501 : WSTRING(55) := " [PIN_239 ]: PvgRightTrackLowside -  HS Short To Ground";
  gc_ErrTranslation_de_Text502 : WSTRING(58) := " [PIN_239 ]: PvgRightTrackLowside -  Internal Driver Error";
  gc_ErrTranslation_de_Text503 : WSTRING(78) := " [PIN_133 PIN_107 ]: FrameRotationSensor1 -  Logical Error between pin 0 and 1";
  gc_ErrTranslation_de_Text504 : WSTRING(63) := " [PIN_133 PIN_107 ]: FrameRotationSensor1 -  Vin0 < u16VolLoMin";
  gc_ErrTranslation_de_Text505 : WSTRING(63) := " [PIN_133 PIN_107 ]: FrameRotationSensor1 -  Vin0 > u16VolHiMax";
  gc_ErrTranslation_de_Text506 : WSTRING(77) := " [PIN_133 PIN_107 ]: FrameRotationSensor1 -  u16VolLoMax < Vin0 < u16VolHiMin";
  gc_ErrTranslation_de_Text507 : WSTRING(63) := " [PIN_133 PIN_107 ]: FrameRotationSensor1 -  Vin1 < u16VolLoMin";
  gc_ErrTranslation_de_Text508 : WSTRING(63) := " [PIN_133 PIN_107 ]: FrameRotationSensor1 -  Vin1 > u16VolHiMax";
  gc_ErrTranslation_de_Text509 : WSTRING(77) := " [PIN_133 PIN_107 ]: FrameRotationSensor1 -  u16VolLoMax < Vin1 < u16VolHiMin";
  gc_ErrTranslation_de_Text510 : WSTRING(78) := " [PIN_114 PIN_112 ]: FrameRotationSensor2 -  Logical Error between pin 0 and 1";
  gc_ErrTranslation_de_Text511 : WSTRING(63) := " [PIN_114 PIN_112 ]: FrameRotationSensor2 -  Vin0 < u16VolLoMin";
  gc_ErrTranslation_de_Text512 : WSTRING(63) := " [PIN_114 PIN_112 ]: FrameRotationSensor2 -  Vin0 > u16VolHiMax";
  gc_ErrTranslation_de_Text513 : WSTRING(77) := " [PIN_114 PIN_112 ]: FrameRotationSensor2 -  u16VolLoMax < Vin0 < u16VolHiMin";
  gc_ErrTranslation_de_Text514 : WSTRING(63) := " [PIN_114 PIN_112 ]: FrameRotationSensor2 -  Vin1 < u16VolLoMin";
  gc_ErrTranslation_de_Text515 : WSTRING(63) := " [PIN_114 PIN_112 ]: FrameRotationSensor2 -  Vin1 > u16VolHiMax";
  gc_ErrTranslation_de_Text516 : WSTRING(77) := " [PIN_114 PIN_112 ]: FrameRotationSensor2 -  u16VolLoMax < Vin1 < u16VolHiMin";
  gc_ErrTranslation_de_Text517 : WSTRING(11) := "Error bit 6";
  gc_ErrTranslation_de_Text518 : WSTRING(11) := "Error bit 7";
  gc_ErrTranslation_de_Text519 : WSTRING(52) := "An input signal is too low / Short circuit to ground";
  gc_ErrTranslation_de_Text520 : WSTRING(52) := "An input signal is too high / Short circuit to power";
  gc_ErrTranslation_de_Text521 : WSTRING(37) := "An input signal is out of valid range";
  gc_ErrTranslation_de_Text522 : WSTRING(39) := "Warning: a block has limited parameters";
  gc_ErrTranslation_de_Text523 : WSTRING(37) := "HS OpenLoad / Short To Power external";
  gc_ErrTranslation_de_Text524 : WSTRING(26) := "HS Short To Power internal";
  gc_ErrTranslation_de_Text525 : WSTRING(18) := "HS Short To Ground";
  gc_ErrTranslation_de_Text526 : WSTRING(21) := "Internal Driver Error";
  gc_ErrTranslation_de_Text527 : WSTRING(37) := "HS OpenLoad / Short To Power external";
  gc_ErrTranslation_de_Text528 : WSTRING(26) := "HS Short To Power internal";
  gc_ErrTranslation_de_Text529 : WSTRING(18) := "HS Short To Ground";
  gc_ErrTranslation_de_Text530 : WSTRING(21) := "Internal Driver Error";
  gc_ErrTranslation_de_Text531 : WSTRING(37) := "HS OpenLoad / Short To Power external";
  gc_ErrTranslation_de_Text532 : WSTRING(26) := "HS Short To Power internal";
  gc_ErrTranslation_de_Text533 : WSTRING(18) := "HS Short To Ground";
  gc_ErrTranslation_de_Text534 : WSTRING(21) := "Internal Driver Error";
  gc_ErrTranslation_de_Text535 : WSTRING(37) := "HS OpenLoad / Short To Power external";
  gc_ErrTranslation_de_Text536 : WSTRING(26) := "HS Short To Power internal";
  gc_ErrTranslation_de_Text537 : WSTRING(18) := "HS Short To Ground";
  gc_ErrTranslation_de_Text538 : WSTRING(21) := "Internal Driver Error";
  gc_ErrTranslation_de_Text539 : WSTRING(23) := "An initialization error";
  gc_ErrTranslation_de_Text540 : WSTRING(34) := "Master input signal short to power";
  gc_ErrTranslation_de_Text541 : WSTRING(35) := "Master input signal short to ground";
  gc_ErrTranslation_de_Text542 : WSTRING(35) := "Parameter of input char NOT monoton";
  gc_ErrTranslation_de_Text543 : WSTRING(22) := "Unknown internal error";
  gc_ErrTranslation_de_Text544 : WSTRING(34) := "Master input signal short to power";
  gc_ErrTranslation_de_Text545 : WSTRING(35) := "Master input signal short to ground";
  gc_ErrTranslation_de_Text546 : WSTRING(35) := "Parameter of input char NOT monoton";
  gc_ErrTranslation_de_Text547 : WSTRING(22) := "Unknown internal error";
  gc_ErrTranslation_de_Text548 : WSTRING(18) := "HS Short To Ground";
  gc_ErrTranslation_de_Text549 : WSTRING(21) := "Internal Driver Error";
  gc_ErrTranslation_de_Text550 : WSTRING(37) := "HS OpenLoad / Short To Power external";
  gc_ErrTranslation_de_Text551 : WSTRING(26) := "HS Short To Power internal";
